C01828=1107.279,258.473,-73.640,-178.368,10.038,149.556
C01829=1107.283,258.225,-73.611,-178.370,10.036,149.556
C01830=1107.288,257.977,-73.582,-178.373,10.033,149.556
C01831=1107.291,257.728,-73.553,-178.376,10.030,149.556
C01832=1107.296,257.480,-73.524,-178.379,10.027,149.556
C01833=1107.300,257.233,-73.495,-178.381,10.025,149.556
C01834=1107.305,256.984,-73.466,-178.384,10.022,149.557
C01835=1107.308,256.736,-73.437,-178.387,10.019,149.556
C01836=1107.313,256.487,-73.409,-178.390,10.016,149.557
C01837=1107.318,256.239,-73.379,-178.393,10.014,149.557
C01838=1107.322,255.991,-73.350,-178.395,10.011,149.557
C01839=1107.325,255.742,-73.322,-178.397,10.009,149.557
C01840=1107.331,255.398,-73.282,-178.401,10.005,149.557
C01841=1107.338,255.055,-73.242,-178.405,10.001,149.557
C01842=1107.343,254.711,-73.202,-178.409,9.998,149.557
C01843=1107.349,254.367,-73.162,-178.413,9.994,149.557
C01844=1107.353,254.119,-73.133,-178.415,9.992,149.557
C01845=1107.358,253.871,-73.105,-178.418,9.989,149.557
C01846=1107.362,253.623,-73.075,-178.421,9.987,149.558
C01847=1107.366,253.374,-73.047,-178.423,9.985,149.558
C01848=1107.371,253.127,-73.018,-178.427,9.982,149.558
C01849=1107.375,252.878,-72.989,-178.429,9.979,149.558
C01850=1107.379,252.629,-72.961,-178.432,9.977,149.558
C01851=1107.383,252.381,-72.932,-178.435,9.975,149.558
C01852=1107.387,252.133,-72.904,-178.438,9.972,149.558
C01853=1107.392,251.885,-72.875,-178.440,9.970,149.559
C01854=1107.396,251.636,-72.846,-178.443,9.968,149.559
C01855=1107.400,251.388,-72.818,-178.446,9.965,149.559
C01856=1107.405,251.140,-72.789,-178.449,9.963,149.559
C01857=1107.408,250.891,-72.760,-178.452,9.960,149.559
C01858=1107.413,250.643,-72.732,-178.455,9.958,149.560
C01859=1107.417,250.394,-72.704,-178.458,9.955,149.560
C01860=1107.421,250.146,-72.675,-178.460,9.953,149.560
C01861=1107.426,249.898,-72.647,-178.463,9.950,149.560
C01862=1107.430,249.649,-72.618,-178.466,9.947,149.560
C01863=1107.435,249.401,-72.590,-178.469,9.945,149.560
C01864=1107.439,249.153,-72.561,-178.472,9.942,149.560
C01865=1107.443,248.905,-72.533,-178.474,9.940,149.560
C01866=1107.448,248.656,-72.504,-178.477,9.937,149.560
C01867=1107.451,248.408,-72.476,-178.480,9.934,149.560
C01868=1107.456,248.159,-72.447,-178.483,9.931,149.561
C01869=1107.460,247.911,-72.420,-178.485,9.928,149.560
C01870=1107.464,247.663,-72.390,-178.488,9.925,149.561
C01871=1107.469,247.415,-72.362,-178.491,9.922,149.560
C01872=1107.473,247.166,-72.334,-178.493,9.919,149.560
C01873=1107.477,246.917,-72.306,-178.496,9.916,149.560
C01874=1107.481,246.670,-72.278,-178.499,9.913,149.560
C01875=1107.486,246.421,-72.249,-178.501,9.910,149.560
C01876=1107.490,246.173,-72.221,-178.503,9.908,149.560
C01877=1107.494,245.924,-72.193,-178.506,9.905,149.560
C01878=1107.499,245.676,-72.165,-178.509,9.902,149.560
C01879=1107.503,245.428,-72.137,-178.511,9.899,149.560
C01880=1107.508,245.179,-72.108,-178.513,9.897,149.560
C01881=1107.512,244.931,-72.080,-178.516,9.894,149.560
C01882=1107.516,244.683,-72.052,-178.519,9.891,149.560
C01883=1107.520,244.434,-72.024,-178.521,9.888,149.560
C01884=1107.524,244.185,-71.995,-178.524,9.886,149.560
C01885=1107.529,243.938,-71.968,-178.527,9.883,149.561
C01886=1107.533,243.689,-71.939,-178.529,9.880,149.560
C01887=1107.537,243.441,-71.911,-178.532,9.877,149.561
C01888=1107.541,243.192,-71.883,-178.534,9.875,149.561
C01889=1107.545,242.944,-71.855,-178.537,9.872,149.561
C01890=1107.550,242.695,-71.827,-178.540,9.870,149.561
C01891=1107.555,242.447,-71.799,-178.542,9.867,149.561
C01892=1107.558,242.235,-71.775,-178.545,9.864,149.561
C01893=1107.562,242.022,-71.752,-178.547,9.862,149.561
C01894=1107.565,241.809,-71.727,-178.549,9.860,149.561
C01895=1107.569,241.597,-71.703,-178.551,9.858,149.561
C01896=1107.572,241.384,-71.680,-178.553,9.856,149.561
C01897=1107.577,241.171,-71.655,-178.555,9.854,149.561
C01898=1107.581,240.959,-71.632,-178.558,9.851,149.561
C01899=1107.584,240.746,-71.608,-178.560,9.849,149.561
C01900=1107.588,240.498,-71.579,-178.563,9.847,149.561
C01901=1107.593,240.249,-71.552,-178.565,9.844,149.561
C01902=1107.596,240.001,-71.524,-178.568,9.841,149.561
C01903=1107.602,239.752,-71.496,-178.570,9.839,149.562
C01904=1107.606,239.503,-71.468,-178.573,9.836,149.562
C01905=1107.610,239.255,-71.441,-178.576,9.833,149.562
C01906=1107.614,239.008,-71.413,-178.579,9.830,149.562
C01907=1107.618,238.759,-71.385,-178.581,9.828,149.562
C01908=1107.623,238.510,-71.358,-178.584,9.826,149.562
C01909=1107.626,238.262,-71.329,-178.587,9.823,149.562
C01910=1107.632,238.013,-71.302,-178.589,9.821,149.562
C01911=1107.636,237.765,-71.274,-178.592,9.818,149.562
C01912=1107.640,237.517,-71.246,-178.595,9.815,149.562
C01913=1107.645,237.268,-71.219,-178.597,9.813,149.562
C01914=1107.648,237.020,-71.191,-178.600,9.810,149.562
C01915=1107.653,236.771,-71.164,-178.603,9.807,149.562
C01916=1107.657,236.523,-71.136,-178.605,9.805,149.563
C01917=1107.661,236.275,-71.108,-178.608,9.802,149.563
C01918=1107.666,236.026,-71.081,-178.611,9.800,149.563
C01919=1107.670,235.778,-71.053,-178.613,9.797,149.563
C01920=1107.674,235.529,-71.025,-178.616,9.795,149.563
C01921=1107.679,235.281,-70.998,-178.619,9.792,149.563
C01922=1107.683,235.033,-70.971,-178.621,9.789,149.563
C01923=1107.687,234.784,-70.942,-178.623,9.787,149.563
C01924=1107.692,234.536,-70.915,-178.626,9.784,149.563
C01925=1107.696,234.287,-70.888,-178.629,9.781,149.563
C01926=1107.700,234.039,-70.860,-178.631,9.779,149.563
C01927=1107.705,233.790,-70.833,-178.634,9.776,149.563
C01928=1107.709,233.542,-70.805,-178.637,9.773,149.563
C01929=1107.713,233.293,-70.778,-178.640,9.771,149.564
C01930=1107.717,233.045,-70.750,-178.642,9.768,149.564
C01931=1107.722,232.797,-70.723,-178.645,9.766,149.564
C01932=1107.726,232.547,-70.696,-178.647,9.763,149.564
C01933=1107.730,232.300,-70.668,-178.650,9.760,149.564
C01934=1107.735,232.051,-70.641,-178.653,9.758,149.564
C01935=1107.740,231.803,-70.614,-178.655,9.755,149.564
C01936=1107.744,231.554,-70.586,-178.658,9.752,149.564
C01937=1107.748,231.305,-70.559,-178.661,9.749,149.564
C01938=1107.753,231.057,-70.532,-178.663,9.747,149.564
C01939=1107.758,230.808,-70.504,-178.665,9.744,149.564
C01940=1107.761,230.560,-70.477,-178.668,9.741,149.564
C01941=1107.765,230.312,-70.450,-178.671,9.738,149.564
C01942=1107.770,230.063,-70.423,-178.674,9.735,149.564
C01943=1107.774,229.815,-70.396,-178.676,9.733,149.564
C01944=1107.778,229.566,-70.368,-178.679,9.730,149.564
C01945=1107.783,229.318,-70.341,-178.681,9.727,149.564
C01946=1107.788,229.069,-70.313,-178.684,9.724,149.564
C01947=1107.791,228.821,-70.287,-178.687,9.721,149.564
C01948=1107.795,228.608,-70.263,-178.689,9.719,149.564
C01949=1107.799,228.395,-70.240,-178.690,9.716,149.564
C01950=1107.803,228.183,-70.217,-178.693,9.714,149.564
C01951=1107.806,227.970,-70.194,-178.695,9.711,149.564
C01952=1107.810,227.757,-70.170,-178.697,9.709,149.564
C01953=1107.814,227.545,-70.147,-178.700,9.706,149.564
C01954=1107.817,227.332,-70.124,-178.702,9.704,149.564
C01955=1107.821,227.119,-70.101,-178.704,9.702,149.564
C01956=1107.826,226.870,-70.074,-178.706,9.699,149.564
C01957=1107.830,226.622,-70.047,-178.709,9.695,149.564
C01958=1107.834,226.374,-70.020,-178.712,9.692,149.564
C01959=1107.838,226.124,-69.993,-178.714,9.689,149.564
C01960=1107.843,225.876,-69.966,-178.716,9.687,149.564
C01961=1107.848,225.627,-69.939,-178.718,9.684,149.564
C01962=1107.852,225.379,-69.912,-178.721,9.681,149.564
C01963=1107.856,225.131,-69.885,-178.723,9.678,149.564
C01964=1107.861,224.882,-69.858,-178.726,9.674,149.563
C01965=1107.865,224.634,-69.832,-178.729,9.671,149.563
C01966=1107.869,224.386,-69.805,-178.731,9.668,149.563
C01967=1107.874,224.136,-69.778,-178.733,9.666,149.563
C01968=1107.878,223.888,-69.751,-178.735,9.663,149.563
C01969=1107.882,223.639,-69.724,-178.738,9.660,149.563
C01970=1107.887,223.391,-69.697,-178.741,9.657,149.563
C01971=1107.891,223.142,-69.671,-178.743,9.653,149.563
C01972=1107.896,222.894,-69.644,-178.746,9.650,149.563
C01973=1107.900,222.646,-69.617,-178.748,9.647,149.563
C01974=1107.904,222.397,-69.590,-178.750,9.645,149.563
C01975=1107.909,222.148,-69.564,-178.753,9.642,149.563
C01976=1107.913,221.900,-69.537,-178.755,9.639,149.563
C01977=1107.918,221.651,-69.510,-178.757,9.635,149.562
C01978=1107.922,221.403,-69.484,-178.760,9.632,149.562
C01979=1107.926,221.155,-69.457,-178.762,9.629,149.562
C01980=1107.931,220.905,-69.430,-178.765,9.626,149.562
C01981=1107.935,220.657,-69.404,-178.767,9.623,149.562
C01982=1107.939,220.408,-69.377,-178.769,9.620,149.562
C01983=1107.943,220.160,-69.350,-178.771,9.617,149.562
C01984=1107.948,219.911,-69.324,-178.774,9.614,149.562
C01985=1107.952,219.663,-69.297,-178.776,9.611,149.562
C01986=1107.957,219.414,-69.270,-178.779,9.608,149.562
C01987=1107.961,219.166,-69.245,-178.781,9.605,149.562
C01988=1107.966,218.917,-69.217,-178.783,9.602,149.561
C01989=1107.970,218.669,-69.191,-178.785,9.599,149.561
C01990=1107.974,218.420,-69.165,-178.788,9.596,149.561
C01991=1107.978,218.172,-69.138,-178.790,9.592,149.561
C01992=1107.982,217.923,-69.112,-178.793,9.589,149.561
C01993=1107.987,217.674,-69.085,-178.794,9.587,149.561
C01994=1107.991,217.426,-69.059,-178.797,9.583,149.561
C01995=1107.996,217.177,-69.033,-178.799,9.580,149.561
C01996=1108.000,216.929,-69.006,-178.802,9.577,149.561
C01997=1108.005,216.680,-68.980,-178.803,9.575,149.560
C01998=1108.009,216.431,-68.953,-178.806,9.571,149.560
C01999=1108.013,216.183,-68.928,-178.808,9.568,149.560
C02000=1108.018,215.935,-68.901,-178.811,9.565,149.560
C02001=1108.023,215.686,-68.875,-178.814,9.562,149.560
C02002=1108.027,215.438,-68.848,-178.815,9.559,149.560
C02003=1108.032,215.189,-68.822,-178.818,9.556,149.560
C02004=1108.035,214.976,-68.799,-178.819,9.554,149.560
C02005=1108.039,214.763,-68.777,-178.821,9.552,149.560
C02006=1108.042,214.550,-68.755,-178.824,9.549,149.560
C02007=1108.046,214.338,-68.732,-178.826,9.546,149.560
C02008=1108.050,214.124,-68.709,-178.827,9.544,149.559
C02009=1108.054,213.912,-68.688,-178.829,9.541,149.559
C02010=1108.057,213.699,-68.665,-178.831,9.539,149.559
C02011=1108.062,213.486,-68.642,-178.834,9.536,149.559
C02012=1108.066,213.237,-68.617,-178.836,9.533,149.559
C02013=1108.070,212.989,-68.590,-178.840,9.529,149.559
C02014=1108.075,212.740,-68.564,-178.842,9.526,149.559
C02015=1108.079,212.491,-68.538,-178.846,9.522,149.559
C02016=1108.083,212.243,-68.511,-178.849,9.520,149.559
C02017=1108.087,211.994,-68.486,-178.852,9.516,149.559
C02018=1108.093,211.746,-68.460,-178.855,9.513,149.559
C02019=1108.097,211.497,-68.433,-178.858,9.509,149.559
C02020=1108.101,211.249,-68.408,-178.861,9.506,149.559
C02021=1108.105,211.000,-68.382,-178.864,9.503,149.560
C02022=1108.110,210.751,-68.355,-178.867,9.500,149.560
C02023=1108.114,210.502,-68.329,-178.871,9.496,149.560
C02024=1108.119,210.254,-68.304,-178.873,9.494,149.560
C02025=1108.123,210.006,-68.278,-178.876,9.491,149.560
C02026=1108.127,209.757,-68.252,-178.880,9.487,149.560
C02027=1108.131,209.508,-68.226,-178.883,9.484,149.560
C02028=1108.136,209.259,-68.200,-178.885,9.481,149.560
C02029=1108.141,209.011,-68.174,-178.889,9.478,149.560
C02030=1108.145,208.763,-68.148,-178.892,9.475,149.560
C02031=1108.149,208.514,-68.122,-178.895,9.472,149.560
C02032=1108.154,208.265,-68.097,-178.897,9.469,149.561
C02033=1108.158,208.017,-68.071,-178.901,9.466,149.561
C02034=1108.163,207.768,-68.045,-178.904,9.463,149.561
C02035=1108.167,207.519,-68.020,-178.907,9.460,149.561
C02036=1108.172,207.270,-67.993,-178.909,9.457,149.561
C02037=1108.177,207.022,-67.968,-178.912,9.454,149.561
C02038=1108.181,206.773,-67.942,-178.915,9.451,149.561
C02039=1108.185,206.524,-67.917,-178.919,9.448,149.561
C02040=1108.189,206.276,-67.891,-178.921,9.445,149.561
C02041=1108.194,206.027,-67.865,-178.924,9.442,149.561
C02042=1108.198,205.779,-67.840,-178.927,9.439,149.561
C02043=1108.203,205.530,-67.814,-178.930,9.436,149.561
C02044=1108.207,205.282,-67.788,-178.933,9.434,149.562
C02045=1108.212,205.033,-67.763,-178.936,9.431,149.562
C02046=1108.216,204.784,-67.738,-178.938,9.428,149.562
C02047=1108.221,204.535,-67.712,-178.941,9.425,149.562
C02048=1108.225,204.287,-67.687,-178.944,9.422,149.562
C02049=1108.229,204.038,-67.661,-178.947,9.420,149.562
C02050=1108.234,203.790,-67.635,-178.950,9.417,149.562
C02051=1108.239,203.541,-67.610,-178.953,9.414,149.562
C02052=1108.243,203.291,-67.585,-178.956,9.411,149.562
C02053=1108.248,203.043,-67.559,-178.958,9.408,149.562
C02054=1108.252,202.795,-67.534,-178.961,9.405,149.562
C02055=1108.256,202.546,-67.508,-178.964,9.402,149.563
C02056=1108.260,202.298,-67.483,-178.967,9.399,149.562
C02057=1108.265,202.049,-67.458,-178.970,9.397,149.563
C02058=1108.269,201.800,-67.432,-178.972,9.393,149.563
C02059=1108.274,201.552,-67.407,-178.975,9.391,149.563
C02060=1108.278,201.338,-67.386,-178.977,9.388,149.563
C02061=1108.281,201.125,-67.363,-178.979,9.386,149.563
C02062=1108.285,200.912,-67.342,-178.982,9.383,149.563
C02063=1108.290,200.699,-67.321,-178.984,9.381,149.563
C02064=1108.293,200.486,-67.298,-178.986,9.379,149.563
C02065=1108.297,200.273,-67.277,-178.988,9.376,149.563
C02066=1108.301,200.060,-67.255,-178.990,9.374,149.563
C02067=1108.304,199.848,-67.234,-178.993,9.372,149.563
C02068=1108.308,199.599,-67.208,-178.995,9.368,149.563
C02069=1108.314,199.350,-67.184,-178.998,9.365,149.563
C02070=1108.318,199.101,-67.158,-179.001,9.363,149.563
C02071=1108.322,198.852,-67.133,-179.003,9.360,149.563
C02072=1108.326,198.604,-67.108,-179.006,9.356,149.563
C02073=1108.331,198.355,-67.083,-179.008,9.353,149.563
C02074=1108.336,198.107,-67.058,-179.010,9.351,149.563
C02075=1108.340,197.857,-67.033,-179.013,9.348,149.563
C02076=1108.344,197.609,-67.008,-179.016,9.345,149.563
C02077=1108.349,197.360,-66.983,-179.018,9.342,149.563
C02078=1108.354,197.112,-66.958,-179.021,9.339,149.563
C02079=1108.358,196.862,-66.932,-179.023,9.336,149.563
C02080=1108.362,196.615,-66.908,-179.025,9.333,149.563
C02081=1108.367,196.365,-66.883,-179.027,9.330,149.562
C02082=1108.372,196.117,-66.857,-179.030,9.327,149.562
C02083=1108.375,195.868,-66.833,-179.032,9.325,149.562
C02084=1108.380,195.620,-66.807,-179.034,9.321,149.562
C02085=1108.385,195.370,-66.782,-179.036,9.318,149.562
C02086=1108.389,195.122,-66.758,-179.038,9.316,149.562
C02087=1108.393,194.873,-66.733,-179.041,9.313,149.562
C02088=1108.399,194.625,-66.708,-179.043,9.310,149.562
C02089=1108.402,194.375,-66.683,-179.045,9.307,149.562
C02090=1108.407,194.127,-66.658,-179.047,9.304,149.562
C02091=1108.411,193.878,-66.634,-179.049,9.301,149.562
C02092=1108.416,193.629,-66.609,-179.052,9.298,149.561
C02093=1108.420,193.381,-66.583,-179.053,9.296,149.561
C02094=1108.425,193.132,-66.559,-179.056,9.293,149.561
C02095=1108.430,192.884,-66.534,-179.058,9.290,149.561
C02096=1108.433,192.635,-66.509,-179.060,9.287,149.561
C02097=1108.438,192.386,-66.485,-179.063,9.284,149.561
C02098=1108.443,192.137,-66.460,-179.065,9.282,149.561
C02099=1108.447,191.888,-66.436,-179.067,9.279,149.561
C02100=1108.452,191.639,-66.411,-179.069,9.276,149.561
C02101=1108.456,191.391,-66.386,-179.071,9.273,149.561
C02102=1108.461,191.143,-66.361,-179.074,9.270,149.561
C02103=1108.465,190.893,-66.337,-179.076,9.267,149.561
C02104=1108.470,190.645,-66.312,-179.078,9.264,149.561
C02105=1108.474,190.396,-66.288,-179.080,9.262,149.561
C02106=1108.479,190.148,-66.262,-179.083,9.259,149.561
C02107=1108.483,189.899,-66.238,-179.085,9.256,149.561
C02108=1108.488,189.650,-66.213,-179.087,9.253,149.561
C02109=1108.492,189.401,-66.189,-179.090,9.250,149.561
C02110=1108.497,189.153,-66.164,-179.092,9.247,149.560
C02111=1108.501,188.903,-66.140,-179.094,9.245,149.560
C02112=1108.506,188.655,-66.115,-179.097,9.242,149.560
C02113=1108.510,188.406,-66.091,-179.098,9.239,149.560
C02114=1108.515,188.157,-66.066,-179.101,9.236,149.560
C02115=1108.519,187.908,-66.042,-179.104,9.234,149.560
C02116=1108.524,187.695,-66.021,-179.106,9.231,149.560
C02117=1108.527,187.483,-66.000,-179.108,9.229,149.560
C02118=1108.531,187.270,-65.979,-179.110,9.227,149.560
C02119=1108.535,187.056,-65.957,-179.111,9.224,149.560
C02120=1108.539,186.843,-65.937,-179.113,9.222,149.560
C02121=1108.543,186.630,-65.916,-179.115,9.220,149.560
C02122=1108.546,186.417,-65.895,-179.117,9.217,149.560
C02123=1108.551,186.204,-65.874,-179.120,9.214,149.560
C02124=1108.554,185.955,-65.850,-179.122,9.212,149.560
C02125=1108.559,185.706,-65.825,-179.124,9.209,149.560
C02126=1108.564,185.458,-65.801,-179.126,9.206,149.560
C02127=1108.568,185.209,-65.777,-179.128,9.203,149.560
C02128=1108.573,184.959,-65.753,-179.131,9.200,149.560
C02129=1108.577,184.711,-65.728,-179.134,9.197,149.560
C02130=1108.582,184.462,-65.704,-179.135,9.195,149.560
C02131=1108.586,184.213,-65.679,-179.138,9.192,149.560
C02132=1108.591,183.965,-65.655,-179.140,9.189,149.560
C02133=1108.595,183.716,-65.631,-179.142,9.186,149.560
C02134=1108.600,183.468,-65.607,-179.145,9.183,149.560
C02135=1108.604,183.218,-65.583,-179.147,9.180,149.560
C02136=1108.609,182.969,-65.559,-179.149,9.178,149.560
C02137=1108.614,182.721,-65.534,-179.151,9.174,149.559
C02138=1108.618,182.472,-65.510,-179.154,9.171,149.559
C02139=1108.622,182.223,-65.486,-179.156,9.168,149.559
C02140=1108.627,181.974,-65.462,-179.158,9.166,149.559
C02141=1108.632,181.725,-65.438,-179.161,9.162,149.559
C02142=1108.636,181.477,-65.413,-179.163,9.159,149.559
C02143=1108.641,181.229,-65.389,-179.166,9.156,149.559
C02144=1108.645,180.979,-65.366,-179.168,9.154,149.559
C02145=1108.649,180.730,-65.342,-179.170,9.151,149.559
C02146=1108.654,180.482,-65.317,-179.173,9.148,149.559
C02147=1108.659,180.233,-65.294,-179.175,9.144,149.559
C02148=1108.663,179.984,-65.269,-179.177,9.142,149.559
C02149=1108.667,179.735,-65.245,-179.179,9.139,149.559
C02150=1108.672,179.486,-65.222,-179.182,9.136,149.559
C02151=1108.676,179.238,-65.198,-179.184,9.132,149.558
C02152=1108.681,178.989,-65.173,-179.186,9.130,149.558
C02153=1108.686,178.740,-65.150,-179.188,9.127,149.558
C02154=1108.691,178.492,-65.126,-179.191,9.124,149.558
C02155=1108.695,178.242,-65.102,-179.192,9.121,149.558
C02156=1108.699,177.993,-65.078,-179.195,9.118,149.558
C02157=1108.703,177.745,-65.054,-179.197,9.115,149.558
C02158=1108.708,177.496,-65.030,-179.199,9.112,149.558
C02159=1108.713,177.248,-65.006,-179.201,9.109,149.558
C02160=1108.717,176.998,-64.983,-179.204,9.106,149.558
C02161=1108.722,176.750,-64.959,-179.205,9.103,149.557
C02162=1108.727,176.500,-64.934,-179.208,9.100,149.557
C02163=1108.731,176.252,-64.910,-179.210,9.097,149.557
C02164=1108.736,176.003,-64.887,-179.212,9.094,149.557
C02165=1108.740,175.754,-64.863,-179.214,9.091,149.557
C02166=1108.745,175.505,-64.840,-179.217,9.088,149.557
C02167=1108.749,175.256,-64.816,-179.218,9.085,149.557
C02168=1108.754,175.008,-64.792,-179.221,9.082,149.557
C02169=1108.758,174.759,-64.769,-179.223,9.079,149.557
C02170=1108.763,174.510,-64.745,-179.225,9.076,149.556
C02171=1108.768,174.261,-64.721,-179.227,9.073,149.556
C02172=1108.771,174.048,-64.701,-179.229,9.071,149.556
C02173=1108.775,173.835,-64.681,-179.231,9.068,149.556
C02174=1108.779,173.621,-64.660,-179.233,9.066,149.556
C02175=1108.783,173.408,-64.640,-179.235,9.064,149.556
C02176=1108.786,173.195,-64.620,-179.237,9.060,149.556
C02177=1108.791,172.982,-64.600,-179.239,9.058,149.556
C02178=1108.795,172.768,-64.580,-179.240,9.055,149.556
C02179=1108.799,172.555,-64.559,-179.242,9.053,149.556
C02180=1108.803,172.306,-64.536,-179.244,9.050,149.555
C02181=1108.808,172.058,-64.512,-179.246,9.047,149.555
C02182=1108.812,171.809,-64.488,-179.249,9.044,149.555
C02183=1108.816,171.560,-64.466,-179.251,9.041,149.555
C02184=1108.821,171.311,-64.442,-179.253,9.038,149.555
C02185=1108.825,171.063,-64.418,-179.255,9.035,149.555
C02186=1108.830,170.814,-64.395,-179.257,9.032,149.555
C02187=1108.835,170.565,-64.372,-179.259,9.029,149.555
C02188=1108.840,170.316,-64.348,-179.262,9.026,149.555
C02189=1108.844,170.067,-64.325,-179.264,9.023,149.554
C02190=1108.849,169.818,-64.301,-179.266,9.020,149.554
C02191=1108.853,169.569,-64.277,-179.268,9.017,149.554
C02192=1108.857,169.320,-64.255,-179.270,9.014,149.554
C02193=1108.862,169.071,-64.231,-179.272,9.012,149.554
C02194=1108.867,168.822,-64.208,-179.275,9.008,149.554
C02195=1108.871,168.573,-64.185,-179.277,9.005,149.554
C02196=1108.876,168.324,-64.161,-179.279,9.003,149.554
C02197=1108.881,168.076,-64.137,-179.281,8.999,149.554
C02198=1108.884,167.827,-64.114,-179.283,8.996,149.553
C02199=1108.889,167.578,-64.091,-179.285,8.994,149.553
C02200=1108.894,167.329,-64.068,-179.287,8.990,149.553
C02201=1108.899,167.081,-64.045,-179.290,8.987,149.553
C02202=1108.904,166.832,-64.021,-179.291,8.984,149.553
C02203=1108.908,166.583,-63.999,-179.294,8.981,149.553
C02204=1108.913,166.334,-63.975,-179.296,8.978,149.553
C02205=1108.917,166.085,-63.952,-179.298,8.975,149.553
C02206=1108.922,165.836,-63.928,-179.300,8.972,149.553
C02207=1108.926,165.587,-63.906,-179.302,8.969,149.552
C02208=1108.931,165.338,-63.882,-179.305,8.966,149.552
C02209=1108.935,165.089,-63.859,-179.306,8.963,149.552
C02210=1108.941,164.841,-63.836,-179.309,8.960,149.552
C02211=1108.945,164.592,-63.813,-179.311,8.956,149.552
C02212=1108.949,164.343,-63.790,-179.314,8.953,149.552
C02213=1108.954,164.094,-63.767,-179.315,8.951,149.552
C02214=1108.958,163.845,-63.744,-179.318,8.947,149.551
C02215=1108.963,163.596,-63.721,-179.320,8.944,149.551
C02216=1108.968,163.347,-63.698,-179.321,8.942,149.551
C02217=1108.972,163.098,-63.675,-179.324,8.939,149.551
C02218=1108.977,162.850,-63.652,-179.326,8.935,149.551
C02219=1108.982,162.600,-63.629,-179.329,8.932,149.551
C02220=1108.986,162.352,-63.606,-179.330,8.929,149.551
C02221=1108.991,162.102,-63.583,-179.333,8.926,149.551
C02222=1108.995,161.853,-63.560,-179.335,8.923,149.550
C02223=1108.999,161.604,-63.537,-179.337,8.920,149.550
C02224=1109.005,161.356,-63.514,-179.339,8.917,149.550
C02225=1109.009,161.107,-63.491,-179.341,8.913,149.550
C02226=1109.014,160.858,-63.469,-179.343,8.910,149.550
C02227=1109.017,160.609,-63.446,-179.345,8.907,149.550
C02228=1109.022,160.396,-63.426,-179.347,8.904,149.550
C02229=1109.026,160.183,-63.407,-179.349,8.902,149.549
C02230=1109.029,159.969,-63.387,-179.351,8.899,149.549
C02231=1109.034,159.756,-63.367,-179.352,8.897,149.549
C02232=1109.038,159.543,-63.348,-179.355,8.894,149.549
C02233=1109.041,159.329,-63.328,-179.356,8.891,149.549
C02234=1109.045,159.116,-63.309,-179.358,8.889,149.549
C02235=1109.049,158.902,-63.290,-179.359,8.886,149.549
C02236=1109.054,158.653,-63.267,-179.362,8.883,149.549
C02237=1109.058,158.405,-63.244,-179.364,8.879,149.548
C02238=1109.063,158.156,-63.222,-179.366,8.876,149.548
C02239=1109.067,157.907,-63.199,-179.369,8.873,149.548
C02240=1109.072,157.658,-63.175,-179.370,8.870,149.548
C02241=1109.077,157.409,-63.154,-179.372,8.866,149.548
C02242=1109.082,157.160,-63.130,-179.375,8.863,149.547
C02243=1109.086,156.911,-63.108,-179.377,8.860,149.547
C02244=1109.091,156.662,-63.085,-179.379,8.856,149.547
C02245=1109.095,156.413,-63.063,-179.380,8.854,149.547
C02246=1109.100,156.164,-63.040,-179.383,8.851,149.547
C02247=1109.104,155.915,-63.017,-179.385,8.847,149.547
C02248=1109.109,155.667,-62.995,-179.387,8.844,149.546
C02249=1109.114,155.418,-62.972,-179.389,8.840,149.546
C02250=1109.118,155.168,-62.950,-179.391,8.838,149.546
C02251=1109.123,154.920,-62.927,-179.393,8.834,149.546
C02252=1109.127,154.671,-62.905,-179.395,8.831,149.546
C02253=1109.132,154.421,-62.883,-179.397,8.827,149.545
C02254=1109.137,154.173,-62.860,-179.399,8.824,149.545
C02255=1109.141,153.924,-62.838,-179.402,8.821,149.545
C02256=1109.146,153.675,-62.815,-179.403,8.818,149.545
C02257=1109.151,153.426,-62.793,-179.405,8.814,149.545
C02258=1109.155,153.177,-62.770,-179.407,8.811,149.544
C02259=1109.160,152.928,-62.747,-179.409,8.807,149.544
C02260=1109.165,152.679,-62.726,-179.412,8.804,149.544
C02261=1109.169,152.430,-62.703,-179.414,8.801,149.544
C02262=1109.174,152.181,-62.681,-179.416,8.797,149.544
C02263=1109.179,151.932,-62.659,-179.418,8.794,149.543
C02264=1109.182,151.683,-62.636,-179.420,8.791,149.543
C02265=1109.187,151.435,-62.614,-179.422,8.788,149.543
C02266=1109.192,151.185,-62.592,-179.424,8.784,149.543
C02267=1109.196,150.936,-62.569,-179.426,8.781,149.542
C02268=1109.201,150.688,-62.547,-179.428,8.777,149.542
C02269=1109.206,150.438,-62.525,-179.430,8.774,149.542
C02270=1109.211,150.189,-62.503,-179.432,8.770,149.542
C02271=1109.215,149.941,-62.480,-179.434,8.767,149.541
C02272=1109.220,149.692,-62.458,-179.436,8.763,149.541
C02273=1109.225,149.442,-62.436,-179.438,8.760,149.541
C02274=1109.230,149.194,-62.414,-179.440,8.756,149.541
C02275=1109.234,148.944,-62.392,-179.442,8.752,149.540
C02276=1109.238,148.696,-62.369,-179.444,8.750,149.540
C02277=1109.243,148.447,-62.348,-179.446,8.746,149.540
C02278=1109.248,148.197,-62.325,-179.448,8.743,149.540
C02279=1109.253,147.949,-62.303,-179.450,8.739,149.539
C02280=1109.257,147.699,-62.281,-179.452,8.736,149.539
C02281=1109.262,147.451,-62.260,-179.454,8.732,149.539
C02282=1109.266,147.201,-62.237,-179.456,8.729,149.539
C02283=1109.271,146.953,-62.215,-179.458,8.725,149.538
C02284=1109.275,146.739,-62.196,-179.460,8.721,149.538
C02285=1109.279,146.526,-62.178,-179.461,8.719,149.538
C02286=1109.283,146.312,-62.158,-179.463,8.716,149.537
C02287=1109.287,146.099,-62.139,-179.465,8.713,149.537
C02288=1109.291,145.886,-62.121,-179.466,8.710,149.537
C02289=1109.295,145.672,-62.102,-179.468,8.706,149.537
C02290=1109.299,145.459,-62.083,-179.470,8.704,149.537
C02291=1109.303,145.245,-62.064,-179.472,8.700,149.536
C02292=1109.308,144.996,-62.043,-179.473,8.697,149.536
C02293=1109.312,144.747,-62.020,-179.475,8.694,149.536
C02294=1109.317,144.498,-61.999,-179.476,8.690,149.535
C02295=1109.321,144.249,-61.977,-179.479,8.686,149.535
C02296=1109.326,144.000,-61.955,-179.480,8.683,149.535
C02297=1109.330,143.751,-61.933,-179.482,8.680,149.534
C02298=1109.335,143.502,-61.911,-179.483,8.676,149.534
C02299=1109.340,143.254,-61.890,-179.485,8.673,149.534
C02300=1109.344,143.004,-61.868,-179.486,8.669,149.533
C02301=1109.349,142.756,-61.846,-179.488,8.666,149.533
C02302=1109.354,142.506,-61.825,-179.491,8.662,149.533
C02303=1109.359,142.257,-61.803,-179.492,8.659,149.532
C02304=1109.363,142.008,-61.781,-179.494,8.656,149.532
C02305=1109.368,141.759,-61.759,-179.495,8.652,149.532
C02306=1109.373,141.510,-61.737,-179.497,8.649,149.531
C02307=1109.377,141.261,-61.715,-179.499,8.646,149.531
C02308=1109.382,141.012,-61.694,-179.500,8.642,149.531
C02309=1109.386,140.762,-61.672,-179.502,8.638,149.530
C02310=1109.391,140.514,-61.651,-179.504,8.635,149.530
C02311=1109.396,140.265,-61.629,-179.506,8.632,149.530
C02312=1109.400,140.016,-61.607,-179.508,8.628,149.530
C02313=1109.405,139.768,-61.586,-179.509,8.625,149.529
C02314=1109.409,139.518,-61.565,-179.511,8.622,149.529
C02315=1109.414,139.269,-61.543,-179.512,8.618,149.528
C02316=1109.419,139.020,-61.521,-179.514,8.614,149.528
C02317=1109.423,138.771,-61.499,-179.516,8.611,149.528
C02318=1109.428,138.522,-61.478,-179.518,8.608,149.528
C02319=1109.433,138.273,-61.457,-179.520,8.604,149.527
C02320=1109.437,138.024,-61.434,-179.521,8.601,149.527
C02321=1109.443,137.774,-61.414,-179.523,8.598,149.527
C02322=1109.447,137.526,-61.392,-179.525,8.594,149.526
C02323=1109.451,137.277,-61.370,-179.526,8.591,149.526
C02324=1109.456,137.028,-61.349,-179.528,8.587,149.526
C02325=1109.461,136.779,-61.328,-179.530,8.584,149.525
C02326=1109.465,136.530,-61.306,-179.531,8.581,149.525
C02327=1109.470,136.280,-61.285,-179.533,8.577,149.525
C02328=1109.475,136.032,-61.264,-179.535,8.574,149.525
C02329=1109.479,135.782,-61.242,-179.537,8.570,149.524
C02330=1109.484,135.533,-61.221,-179.538,8.567,149.524
C02331=1109.489,135.285,-61.199,-179.540,8.564,149.524
C02332=1109.494,135.035,-61.178,-179.542,8.560,149.523
C02333=1109.498,134.786,-61.157,-179.544,8.558,149.523
C02334=1109.503,134.537,-61.136,-179.545,8.554,149.523
C02335=1109.508,134.289,-61.114,-179.547,8.550,149.523
C02336=1109.512,134.039,-61.093,-179.549,8.548,149.522
C02337=1109.516,133.790,-61.071,-179.550,8.544,149.522
C02338=1109.522,133.541,-61.050,-179.553,8.540,149.522
C02339=1109.526,133.292,-61.029,-179.554,8.537,149.521
C02340=1109.530,133.078,-61.010,-179.556,8.534,149.521
C02341=1109.534,132.865,-60.993,-179.558,8.531,149.521
C02342=1109.538,132.652,-60.975,-179.559,8.529,149.521
C02343=1109.543,132.438,-60.956,-179.560,8.525,149.520
C02344=1109.546,132.224,-60.938,-179.561,8.523,149.520
C02345=1109.550,132.010,-60.920,-179.563,8.520,149.520
C02346=1109.554,131.797,-60.902,-179.564,8.517,149.520
C02347=1109.558,131.584,-60.884,-179.566,8.514,149.519
C02348=1109.563,131.335,-60.863,-179.568,8.511,149.519
C02349=1109.568,131.085,-60.841,-179.570,8.508,149.519
C02350=1109.572,130.837,-60.820,-179.572,8.504,149.518
C02351=1109.577,130.587,-60.800,-179.573,8.501,149.518
C02352=1109.582,130.339,-60.778,-179.575,8.498,149.518
C02353=1109.586,130.090,-60.757,-179.577,8.494,149.518
C02354=1109.591,129.840,-60.736,-179.578,8.491,149.517
C02355=1109.596,129.591,-60.714,-179.580,8.487,149.517
C02356=1109.600,129.342,-60.694,-179.582,8.484,149.517
C02357=1109.606,129.093,-60.673,-179.584,8.481,149.517
C02358=1109.610,128.845,-60.652,-179.585,8.477,149.516
C02359=1109.615,128.595,-60.631,-179.587,8.474,149.516
C02360=1109.619,128.345,-60.610,-179.589,8.471,149.516
C02361=1109.624,128.096,-60.589,-179.591,8.468,149.516
C02362=1109.629,127.848,-60.568,-179.592,8.464,149.515
C02363=1109.633,127.599,-60.547,-179.594,8.461,149.515
C02364=1109.638,127.350,-60.526,-179.596,8.458,149.515
C02365=1109.644,127.100,-60.505,-179.598,8.454,149.514
C02366=1109.648,126.852,-60.484,-179.600,8.450,149.514
C02367=1109.652,126.602,-60.463,-179.601,8.447,149.514
C02368=1109.657,126.353,-60.443,-179.603,8.444,149.514
C02369=1109.662,126.104,-60.422,-179.605,8.440,149.513
C02370=1109.666,125.855,-60.401,-179.606,8.437,149.513
C02371=1109.671,125.606,-60.380,-179.608,8.434,149.513
C02372=1109.676,125.357,-60.359,-179.610,8.430,149.512
C02373=1109.681,125.108,-60.338,-179.612,8.428,149.512
C02374=1109.685,124.859,-60.318,-179.613,8.424,149.512
C02375=1109.690,124.610,-60.297,-179.616,8.420,149.511
C02376=1109.694,124.360,-60.276,-179.617,8.418,149.511
C02377=1109.699,124.111,-60.256,-179.619,8.414,149.511
C02378=1109.704,123.862,-60.235,-179.621,8.410,149.511
C02379=1109.708,123.613,-60.214,-179.622,8.407,149.510
C02380=1109.713,123.364,-60.193,-179.624,8.404,149.510
C02381=1109.718,123.115,-60.173,-179.626,8.400,149.510
C02382=1109.723,122.865,-60.152,-179.627,8.397,149.509
C02383=1109.727,122.617,-60.132,-179.629,8.394,149.509
C02384=1109.732,122.368,-60.111,-179.631,8.390,149.509
C02385=1109.737,122.118,-60.090,-179.633,8.387,149.509
C02386=1109.742,121.869,-60.070,-179.634,8.384,149.508
C02387=1109.747,121.620,-60.049,-179.636,8.380,149.508
C02388=1109.751,121.371,-60.029,-179.639,8.377,149.508
C02389=1109.756,121.122,-60.008,-179.640,8.374,149.508
C02390=1109.761,120.873,-59.987,-179.642,8.370,149.507
C02391=1109.765,120.624,-59.967,-179.644,8.367,149.507
C02392=1109.770,120.375,-59.947,-179.645,8.364,149.507
C02393=1109.775,120.126,-59.926,-179.647,8.360,149.507
C02394=1109.779,119.877,-59.905,-179.649,8.357,149.506
C02395=1109.784,119.628,-59.885,-179.650,8.354,149.506
C02396=1109.788,119.414,-59.868,-179.652,8.350,149.506
C02397=1109.792,119.200,-59.850,-179.654,8.348,149.505
C02398=1109.796,118.987,-59.833,-179.655,8.345,149.505
C02399=1109.800,118.773,-59.815,-179.657,8.342,149.505
C02400=1109.804,118.559,-59.797,-179.658,8.340,149.505
C02401=1109.808,118.345,-59.779,-179.660,8.336,149.505
C02402=1109.812,118.132,-59.763,-179.662,8.333,149.504
C02403=1109.816,117.918,-59.745,-179.663,8.330,149.504
C02404=1109.820,117.669,-59.725,-179.665,8.327,149.504
C02405=1109.826,117.420,-59.704,-179.666,8.324,149.503
C02406=1109.831,117.171,-59.684,-179.668,8.320,149.503
C02407=1109.835,116.922,-59.663,-179.670,8.317,149.503
C02408=1109.840,116.673,-59.644,-179.671,8.314,149.503
C02409=1109.845,116.424,-59.623,-179.673,8.310,149.502
C02410=1109.849,116.175,-59.602,-179.675,8.307,149.502
C02411=1109.854,115.925,-59.583,-179.677,8.303,149.502
C02412=1109.859,115.676,-59.562,-179.678,8.300,149.501
C02413=1109.864,115.427,-59.541,-179.680,8.296,149.501
C02414=1109.868,115.178,-59.521,-179.682,8.293,149.501
C02415=1109.873,114.928,-59.501,-179.683,8.290,149.501
C02416=1109.877,114.679,-59.481,-179.685,8.287,149.500
C02417=1109.882,114.430,-59.461,-179.687,8.283,149.500
C02418=1109.887,114.182,-59.441,-179.689,8.279,149.500
C02419=1109.892,113.932,-59.420,-179.691,8.277,149.499
C02420=1109.897,113.683,-59.401,-179.692,8.273,149.499
C02421=1109.902,113.434,-59.380,-179.694,8.269,149.499
C02422=1109.906,113.185,-59.360,-179.696,8.266,149.499
C02423=1109.911,112.935,-59.340,-179.697,8.263,149.498
C02424=1109.915,112.686,-59.320,-179.699,8.259,149.498
C02425=1109.921,112.438,-59.301,-179.701,8.255,149.497
C02426=1109.926,112.188,-59.280,-179.703,8.252,149.497
C02427=1109.930,111.939,-59.260,-179.704,8.249,149.497
C02428=1109.935,111.690,-59.240,-179.706,8.245,149.497
C02429=1109.940,111.440,-59.220,-179.708,8.242,149.496
C02430=1109.944,111.191,-59.200,-179.710,8.238,149.496
C02431=1109.949,110.942,-59.180,-179.711,8.235,149.496
C02432=1109.954,110.693,-59.160,-179.713,8.232,149.495
C02433=1109.959,110.444,-59.140,-179.716,8.227,149.495
C02434=1109.963,110.195,-59.120,-179.718,8.224,149.495
C02435=1109.968,109.945,-59.100,-179.720,8.220,149.495
C02436=1109.973,109.697,-59.080,-179.722,8.216,149.494
C02437=1109.978,109.447,-59.061,-179.724,8.213,149.494
C02438=1109.982,109.199,-59.040,-179.725,8.209,149.494
C02439=1109.987,108.949,-59.021,-179.727,8.205,149.493
C02440=1109.992,108.700,-59.001,-179.729,8.202,149.493
C02441=1109.997,108.451,-58.981,-179.731,8.198,149.493
C02442=1110.001,108.202,-58.961,-179.733,8.195,149.493
C02443=1110.006,107.952,-58.942,-179.735,8.191,149.492
C02444=1110.010,107.703,-58.921,-179.737,8.187,149.492
C02445=1110.016,107.454,-58.902,-179.739,8.184,149.492
C02446=1110.021,107.205,-58.882,-179.740,8.180,149.491
C02447=1110.025,106.956,-58.862,-179.742,8.176,149.491
C02448=1110.030,106.707,-58.843,-179.744,8.172,149.491
C02449=1110.035,106.457,-58.823,-179.746,8.169,149.490
C02450=1110.039,106.208,-58.803,-179.748,8.165,149.490
C02451=1110.044,105.959,-58.783,-179.750,8.162,149.490
C02452=1110.048,105.745,-58.766,-179.751,8.159,149.489
C02453=1110.053,105.532,-58.750,-179.753,8.155,149.489
C02454=1110.056,105.318,-58.733,-179.754,8.152,149.489
C02455=1110.061,105.104,-58.716,-179.756,8.149,149.489
C02456=1110.064,104.890,-58.700,-179.757,8.146,149.488
C02457=1110.069,104.676,-58.682,-179.759,8.143,149.488
C02458=1110.073,104.462,-58.666,-179.761,8.139,149.488
C02459=1110.077,104.249,-58.649,-179.762,8.136,149.487
C02460=1110.082,104.000,-58.629,-179.764,8.133,149.487
C02461=1110.086,103.750,-58.610,-179.765,8.129,149.487
C02462=1110.091,103.501,-58.590,-179.767,8.125,149.486
C02463=1110.096,103.253,-58.571,-179.769,8.121,149.486
C02464=1110.101,103.003,-58.551,-179.771,8.118,149.485
C02465=1110.106,102.754,-58.532,-179.772,8.114,149.485
C02466=1110.110,102.505,-58.513,-179.774,8.110,149.485
C02467=1110.115,102.255,-58.493,-179.776,8.106,149.484
C02468=1110.120,102.006,-58.474,-179.778,8.102,149.484
C02469=1110.125,101.757,-58.454,-179.779,8.099,149.484
C02470=1110.130,101.507,-58.434,-179.780,8.095,149.483
C02471=1110.134,101.259,-58.416,-179.782,8.092,149.483
C02472=1110.139,101.009,-58.396,-179.784,8.088,149.482
C02473=1110.144,100.760,-58.377,-179.785,8.084,149.482
C02474=1110.148,100.511,-58.358,-179.787,8.080,149.482
C02475=1110.153,100.262,-58.338,-179.789,8.076,149.481
C02476=1110.158,100.013,-58.319,-179.790,8.073,149.481
C02477=1110.163,99.763,-58.299,-179.792,8.069,149.480
C02478=1110.168,99.515,-58.280,-179.794,8.065,149.480
C02479=1110.172,99.265,-58.261,-179.795,8.061,149.480
C02480=1110.177,99.015,-58.241,-179.797,8.057,149.479
C02481=1110.182,98.767,-58.222,-179.799,8.053,149.479
C02482=1110.187,98.517,-58.203,-179.800,8.050,149.478
C02483=1110.192,98.268,-58.183,-179.801,8.046,149.478
C02484=1110.196,98.019,-58.164,-179.803,8.043,149.477
C02485=1110.201,97.770,-58.145,-179.804,8.039,149.477
C02486=1110.206,97.521,-58.125,-179.806,8.035,149.477
C02487=1110.211,97.272,-58.107,-179.808,8.031,149.476
C02488=1110.216,97.022,-58.088,-179.809,8.027,149.476
C02489=1110.220,96.772,-58.068,-179.811,8.023,149.475
C02490=1110.225,96.524,-58.049,-179.812,8.020,149.475
C02491=1110.230,96.274,-58.030,-179.813,8.016,149.474
C02492=1110.234,96.026,-58.011,-179.815,8.012,149.474
C02493=1110.239,95.776,-57.992,-179.817,8.008,149.473
C02494=1110.245,95.527,-57.973,-179.818,8.004,149.473
C02495=1110.249,95.277,-57.954,-179.820,8.001,149.473
C02496=1110.254,95.029,-57.934,-179.821,7.997,149.472
C02497=1110.258,94.779,-57.916,-179.822,7.994,149.472
C02498=1110.264,94.530,-57.897,-179.824,7.990,149.471
C02499=1110.268,94.281,-57.878,-179.826,7.986,149.471
C02500=1110.273,94.032,-57.858,-179.827,7.982,149.470
C02501=1110.277,93.782,-57.840,-179.828,7.978,149.470
C02502=1110.283,93.533,-57.821,-179.829,7.975,149.469
C02503=1110.287,93.284,-57.802,-179.831,7.971,149.469
C02504=1110.292,93.034,-57.783,-179.833,7.967,149.469
C02505=1110.297,92.786,-57.764,-179.834,7.963,149.468
C02506=1110.302,92.536,-57.745,-179.836,7.959,149.468
C02507=1110.307,92.287,-57.727,-179.836,7.956,149.467
C02508=1110.311,92.072,-57.710,-179.838,7.952,149.467
C02509=1110.315,91.859,-57.693,-179.839,7.949,149.466
C02510=1110.319,91.646,-57.678,-179.840,7.946,149.466
C02511=1110.323,91.432,-57.662,-179.841,7.943,149.465
C02512=1110.327,91.217,-57.645,-179.843,7.939,149.465
C02513=1110.332,91.004,-57.629,-179.844,7.936,149.465
C02514=1110.336,90.790,-57.613,-179.845,7.933,149.464
C02515=1110.340,90.576,-57.597,-179.846,7.929,149.464
C02516=1110.344,90.327,-57.578,-179.847,7.926,149.463
C02517=1110.350,90.077,-57.560,-179.849,7.922,149.463
C02518=1110.354,89.828,-57.541,-179.849,7.918,149.462
C02519=1110.360,89.579,-57.522,-179.851,7.914,149.462
C02520=1110.364,89.329,-57.503,-179.853,7.910,149.461
C02521=1110.368,89.080,-57.485,-179.854,7.906,149.461
C02522=1110.374,88.831,-57.466,-179.855,7.903,149.460
C02523=1110.378,88.582,-57.447,-179.856,7.899,149.460
C02524=1110.383,88.333,-57.429,-179.858,7.895,149.459
C02525=1110.388,88.084,-57.410,-179.858,7.892,149.459
C02526=1110.392,87.834,-57.391,-179.860,7.888,149.458
C02527=1110.398,87.585,-57.372,-179.861,7.884,149.458
C02528=1110.403,87.336,-57.354,-179.863,7.880,149.457
C02529=1110.407,87.086,-57.335,-179.864,7.877,149.457
C02530=1110.412,86.837,-57.316,-179.865,7.872,149.456
C02531=1110.417,86.588,-57.298,-179.866,7.868,149.456
C02532=1110.421,86.338,-57.280,-179.867,7.865,149.455
C02533=1110.427,86.090,-57.260,-179.868,7.861,149.455
C02534=1110.432,85.840,-57.242,-179.870,7.857,149.454
C02535=1110.436,85.590,-57.224,-179.871,7.854,149.454
C02536=1110.441,85.342,-57.205,-179.872,7.850,149.453
C02537=1110.446,85.092,-57.187,-179.874,7.846,149.453
C02538=1110.451,84.843,-57.168,-179.874,7.842,149.452
C02539=1110.455,84.594,-57.150,-179.876,7.838,149.452
C02540=1110.460,84.345,-57.132,-179.876,7.835,149.451
C02541=1110.465,84.095,-57.113,-179.878,7.831,149.451
C02542=1110.470,83.846,-57.094,-179.879,7.827,149.450
C02543=1110.475,83.597,-57.076,-179.880,7.824,149.449
C02544=1110.480,83.348,-57.058,-179.881,7.819,149.449
C02545=1110.484,83.098,-57.039,-179.882,7.816,149.448
C02546=1110.489,82.849,-57.021,-179.883,7.812,149.448
C02547=1110.494,82.600,-57.003,-179.885,7.808,149.447
C02548=1110.498,82.350,-56.984,-179.885,7.805,149.447
C02549=1110.504,82.101,-56.965,-179.887,7.801,149.446
C02550=1110.509,81.852,-56.947,-179.888,7.798,149.446
C02551=1110.514,81.603,-56.929,-179.889,7.793,149.445
C02552=1110.518,81.353,-56.911,-179.890,7.790,149.444
C02553=1110.523,81.104,-56.893,-179.891,7.786,149.444
C02554=1110.527,80.855,-56.874,-179.892,7.782,149.443
C02555=1110.533,80.606,-56.855,-179.893,7.779,149.443
C02556=1110.537,80.356,-56.837,-179.894,7.774,149.442
C02557=1110.542,80.107,-56.819,-179.895,7.771,149.442
C02558=1110.547,79.857,-56.801,-179.896,7.767,149.441
C02559=1110.552,79.608,-56.783,-179.897,7.764,149.441
C02560=1110.557,79.359,-56.765,-179.899,7.759,149.440
C02561=1110.561,79.110,-56.746,-179.900,7.756,149.440
C02562=1110.567,78.860,-56.728,-179.901,7.752,149.439
C02563=1110.572,78.611,-56.710,-179.902,7.749,149.439
C02564=1110.576,78.396,-56.694,-179.902,7.745,149.438
C02565=1110.579,78.183,-56.679,-179.903,7.742,149.438
C02566=1110.584,77.970,-56.663,-179.904,7.739,149.437
C02567=1110.588,77.755,-56.648,-179.905,7.736,149.437
C02568=1110.592,77.542,-56.632,-179.906,7.733,149.436
C02569=1110.596,77.328,-56.616,-179.906,7.730,149.436
C02570=1110.601,77.114,-56.601,-179.907,7.726,149.435
C02571=1110.605,76.900,-56.585,-179.908,7.723,149.435
C02572=1110.610,76.650,-56.567,-179.910,7.719,149.434
C02573=1110.615,76.401,-56.549,-179.911,7.715,149.434
C02574=1110.620,76.152,-56.531,-179.913,7.711,149.433
C02575=1110.624,75.902,-56.513,-179.914,7.707,149.433
C02576=1110.629,75.653,-56.495,-179.915,7.704,149.432
C02577=1110.634,75.404,-56.477,-179.916,7.700,149.432
C02578=1110.639,75.155,-56.459,-179.918,7.696,149.431
C02579=1110.644,74.906,-56.441,-179.919,7.692,149.431
C02580=1110.648,74.656,-56.423,-179.921,7.688,149.430
C02581=1110.654,74.407,-56.405,-179.922,7.684,149.430
C02582=1110.659,74.157,-56.388,-179.924,7.680,149.429
C02583=1110.663,73.907,-56.369,-179.925,7.676,149.429
C02584=1110.668,73.658,-56.351,-179.926,7.672,149.428
C02585=1110.673,73.409,-56.333,-179.928,7.668,149.428
C02586=1110.678,73.160,-56.315,-179.930,7.664,149.427
C02587=1110.683,72.911,-56.297,-179.931,7.660,149.427
C02588=1110.687,72.662,-56.279,-179.932,7.657,149.426
C02589=1110.692,72.412,-56.261,-179.933,7.653,149.426
C02590=1110.698,72.163,-56.244,-179.934,7.648,149.425
C02591=1110.702,71.913,-56.226,-179.936,7.645,149.425
C02592=1110.707,71.665,-56.209,-179.937,7.641,149.424
C02593=1110.712,71.415,-56.191,-179.939,7.637,149.424
C02594=1110.716,71.166,-56.172,-179.940,7.632,149.423
C02595=1110.721,70.916,-56.155,-179.942,7.629,149.423
C02596=1110.726,70.667,-56.137,-179.943,7.625,149.422
C02597=1110.731,70.417,-56.119,-179.944,7.620,149.422
C02598=1110.736,70.168,-56.101,-179.945,7.617,149.421
C02599=1110.741,69.918,-56.084,-179.947,7.613,149.421
C02600=1110.746,69.669,-56.066,-179.948,7.609,149.420
C02601=1110.750,69.420,-56.049,-179.950,7.605,149.420
C02602=1110.755,69.171,-56.031,-179.951,7.601,149.419
C02603=1110.760,68.921,-56.013,-179.952,7.597,149.419
C02604=1110.765,68.672,-55.995,-179.954,7.593,149.418
C02605=1110.770,68.422,-55.978,-179.955,7.589,149.418
C02606=1110.775,68.174,-55.961,-179.956,7.586,149.417
C02607=1110.779,67.924,-55.943,-179.958,7.582,149.417
C02608=1110.785,67.675,-55.925,-179.959,7.578,149.416
C02609=1110.790,67.425,-55.907,-179.960,7.574,149.416
C02610=1110.794,67.176,-55.889,-179.962,7.570,149.415
C02611=1110.799,66.927,-55.873,-179.963,7.565,149.415
C02612=1110.804,66.678,-55.855,-179.964,7.561,149.414
C02613=1110.809,66.428,-55.838,-179.966,7.558,149.414
C02614=1110.814,66.179,-55.820,-179.967,7.554,149.413
C02615=1110.818,65.930,-55.802,-179.968,7.550,149.413
C02616=1110.823,65.680,-55.785,-179.970,7.546,149.412
C02617=1110.828,65.431,-55.767,-179.971,7.542,149.412
C02618=1110.834,65.181,-55.750,-179.972,7.538,149.411
C02619=1110.838,64.932,-55.732,-179.973,7.534,149.410
C02620=1110.842,64.718,-55.717,-179.974,7.531,149.410
C02621=1110.846,64.504,-55.703,-179.975,7.528,149.410
C02622=1110.851,64.290,-55.688,-179.977,7.524,149.409
C02623=1110.855,64.076,-55.672,-179.978,7.521,149.409
C02624=1110.859,63.862,-55.658,-179.979,7.517,149.408
C02625=1110.864,63.648,-55.643,-179.980,7.513,149.408
C02626=1110.867,63.434,-55.628,-179.981,7.510,149.407
C02627=1110.872,63.220,-55.613,-179.982,7.507,149.407
C02628=1110.876,62.971,-55.596,-179.983,7.503,149.406
C02629=1110.882,62.721,-55.579,-179.985,7.499,149.406
C02630=1110.886,62.472,-55.561,-179.986,7.495,149.405
C02631=1110.891,62.223,-55.544,-179.988,7.491,149.405
C02632=1110.896,61.974,-55.526,-179.989,7.487,149.404
C02633=1110.901,61.724,-55.510,-179.990,7.483,149.404
C02634=1110.906,61.474,-55.492,-179.991,7.480,149.403
C02635=1110.911,61.225,-55.474,-179.992,7.475,149.403
C02636=1110.915,60.976,-55.458,-179.994,7.471,149.402
C02637=1110.921,60.726,-55.440,-179.995,7.467,149.402
C02638=1110.925,60.477,-55.423,-179.996,7.463,149.401
C02639=1110.931,60.228,-55.406,-179.997,7.460,149.401
C02640=1110.936,59.978,-55.389,-179.999,7.456,149.400
C02641=1110.940,59.729,-55.371,180.000,7.452,149.400
C02642=1110.945,59.480,-55.354,179.999,7.448,149.399
C02643=1110.950,59.230,-55.338,179.997,7.444,149.399
C02644=1110.955,58.980,-55.320,179.996,7.439,149.398
C02645=1110.960,58.732,-55.303,179.995,7.436,149.397
C02646=1110.965,58.482,-55.286,179.994,7.432,149.397
C02647=1110.969,58.233,-55.269,179.993,7.428,149.396
C02648=1110.975,57.983,-55.252,179.991,7.424,149.396
C02649=1110.979,57.734,-55.235,179.990,7.420,149.395
C02650=1110.985,57.485,-55.218,179.989,7.415,149.395
C02651=1110.989,57.236,-55.201,179.988,7.412,149.394
C02652=1110.994,56.986,-55.184,179.987,7.408,149.394
C02653=1110.999,56.736,-55.167,179.985,7.404,149.393
C02654=1111.004,56.487,-55.149,179.984,7.400,149.392
C02655=1111.009,56.238,-55.133,179.983,7.396,149.392
C02656=1111.014,55.989,-55.116,179.981,7.392,149.391
C02657=1111.019,55.739,-55.099,179.981,7.388,149.391
C02658=1111.024,55.489,-55.082,179.979,7.384,149.390
C02659=1111.029,55.241,-55.065,179.978,7.380,149.390
C02660=1111.034,54.991,-55.048,179.977,7.376,149.389
C02661=1111.039,54.741,-55.031,179.976,7.372,149.389
C02662=1111.043,54.492,-55.014,179.974,7.368,149.388
C02663=1111.049,54.243,-54.997,179.974,7.364,149.387
C02664=1111.053,53.994,-54.981,179.972,7.360,149.387
C02665=1111.058,53.744,-54.963,179.971,7.356,149.386
C02666=1111.063,53.495,-54.947,179.970,7.352,149.386
C02667=1111.068,53.246,-54.930,179.968,7.348,149.385
C02668=1111.073,52.996,-54.913,179.968,7.344,149.385
C02669=1111.078,52.746,-54.896,179.966,7.340,149.384
C02670=1111.083,52.497,-54.879,179.965,7.336,149.384
C02671=1111.088,52.248,-54.863,179.964,7.332,149.383
C02672=1111.092,51.998,-54.846,179.963,7.328,149.382
C02673=1111.098,51.749,-54.829,179.962,7.324,149.382
C02674=1111.103,51.500,-54.813,179.961,7.321,149.381
C02675=1111.107,51.250,-54.796,179.959,7.316,149.381
C02676=1111.112,51.036,-54.782,179.959,7.313,149.380
C02677=1111.116,50.822,-54.767,179.957,7.309,149.380
C02678=1111.120,50.608,-54.753,179.957,7.306,149.379
C02679=1111.124,50.394,-54.739,179.956,7.303,149.379
C02680=1111.129,50.180,-54.724,179.954,7.299,149.378
C02681=1111.133,49.966,-54.710,179.954,7.295,149.378
C02682=1111.137,49.751,-54.695,179.953,7.292,149.377
C02683=1111.141,49.537,-54.682,179.952,7.289,149.377
C02684=1111.146,49.288,-54.665,179.951,7.285,149.376
C02685=1111.151,49.038,-54.648,179.950,7.280,149.376
C02686=1111.156,48.789,-54.632,179.948,7.276,149.375
C02687=1111.161,48.540,-54.615,179.947,7.272,149.374
C02688=1111.165,48.291,-54.599,179.946,7.269,149.374
C02689=1111.172,48.041,-54.582,179.945,7.265,149.373
C02690=1111.176,47.791,-54.566,179.944,7.260,149.373
C02691=1111.181,47.542,-54.549,179.943,7.256,149.372
C02692=1111.186,47.293,-54.533,179.941,7.252,149.372
C02693=1111.190,47.044,-54.516,179.941,7.249,149.371
C02694=1111.196,46.793,-54.500,179.940,7.244,149.370
C02695=1111.201,46.544,-54.483,179.939,7.240,149.370
C02696=1111.205,46.295,-54.467,179.937,7.236,149.369
C02697=1111.210,46.046,-54.450,179.936,7.232,149.369
C02698=1111.215,45.796,-54.434,179.935,7.228,149.368
C02699=1111.220,45.547,-54.418,179.934,7.224,149.367
C02700=1111.225,45.298,-54.401,179.933,7.220,149.367
C02701=1111.230,45.047,-54.385,179.932,7.216,149.366
C02702=1111.235,44.799,-54.368,179.931,7.211,149.366
C02703=1111.240,44.549,-54.352,179.930,7.208,149.365
C02704=1111.245,44.300,-54.336,179.929,7.204,149.364
C02705=1111.250,44.050,-54.320,179.928,7.200,149.364
C02706=1111.255,43.801,-54.303,179.927,7.195,149.363
C02707=1111.260,43.551,-54.287,179.925,7.191,149.363
C02708=1111.265,43.302,-54.270,179.925,7.188,149.362
C02709=1111.270,43.053,-54.254,179.923,7.184,149.361
C02710=1111.274,42.803,-54.238,179.922,7.179,149.361
C02711=1111.280,42.554,-54.221,179.921,7.175,149.360
C02712=1111.284,42.304,-54.206,179.920,7.171,149.359
C02713=1111.289,42.055,-54.189,179.920,7.167,149.359
C02714=1111.294,41.806,-54.173,179.918,7.163,149.358
C02715=1111.299,41.556,-54.157,179.917,7.159,149.358
C02716=1111.304,41.307,-54.140,179.916,7.155,149.357
C02717=1111.309,41.057,-54.125,179.915,7.150,149.356
C02718=1111.314,40.808,-54.108,179.915,7.147,149.356
C02719=1111.319,40.558,-54.092,179.913,7.143,149.355
C02720=1111.324,40.309,-54.076,179.912,7.138,149.354
C02721=1111.329,40.059,-54.060,179.911,7.134,149.354
C02722=1111.334,39.811,-54.044,179.910,7.130,149.353
C02723=1111.339,39.561,-54.028,179.909,7.127,149.353
C02724=1111.344,39.312,-54.012,179.908,7.122,149.352
C02725=1111.349,39.062,-53.996,179.907,7.118,149.351
C02726=1111.354,38.813,-53.979,179.906,7.114,149.351
C02727=1111.358,38.563,-53.963,179.906,7.110,149.350
C02728=1111.364,38.313,-53.948,179.905,7.106,149.349
C02729=1111.368,38.064,-53.931,179.904,7.102,149.349
C02730=1111.374,37.815,-53.916,179.902,7.097,149.348
C02731=1111.379,37.566,-53.899,179.901,7.093,149.347
C02732=1111.383,37.351,-53.886,179.900,7.090,149.347
C02733=1111.387,37.137,-53.872,179.900,7.086,149.346
C02734=1111.392,36.923,-53.858,179.899,7.083,149.346
C02735=1111.396,36.708,-53.844,179.898,7.079,149.345
C02736=1111.400,36.494,-53.831,179.897,7.076,149.345
C02737=1111.405,36.280,-53.817,179.897,7.072,149.344
C02738=1111.409,36.065,-53.803,179.896,7.069,149.344
C02739=1111.413,35.851,-53.790,179.895,7.065,149.343
C02740=1111.418,35.603,-53.774,179.894,7.060,149.342
C02741=1111.422,35.353,-53.758,179.893,7.057,149.342
C02742=1111.428,35.103,-53.742,179.892,7.053,149.341
C02743=1111.433,34.854,-53.727,179.891,7.048,149.341
C02744=1111.438,34.604,-53.710,179.890,7.044,149.340
C02745=1111.443,34.355,-53.695,179.889,7.040,149.339
C02746=1111.448,34.105,-53.679,179.888,7.036,149.339
C02747=1111.453,33.855,-53.663,179.887,7.032,149.338
C02748=1111.457,33.607,-53.647,179.886,7.028,149.337
C02749=1111.463,33.358,-53.632,179.885,7.023,149.337
C02750=1111.468,33.107,-53.616,179.885,7.020,149.336
C02751=1111.473,32.858,-53.600,179.884,7.015,149.335
C02752=1111.478,32.609,-53.583,179.883,7.011,149.334
C02753=1111.482,32.359,-53.568,179.882,7.006,149.334
C02754=1111.488,32.110,-53.553,179.881,7.002,149.333
C02755=1111.493,31.861,-53.537,179.881,6.999,149.332
C02756=1111.498,31.611,-53.521,179.880,6.994,149.332
C02757=1111.503,31.361,-53.506,179.879,6.990,149.331
C02758=1111.507,31.113,-53.490,179.877,6.986,149.330
C02759=1111.512,30.863,-53.474,179.876,6.981,149.330
C02760=1111.518,30.613,-53.458,179.876,6.977,149.329
C02761=1111.523,30.364,-53.443,179.875,6.973,149.328
C02762=1111.527,30.114,-53.428,179.874,6.969,149.328
C02763=1111.532,29.865,-53.412,179.873,6.965,149.327
C02764=1111.538,29.615,-53.396,179.872,6.960,149.326
C02765=1111.543,29.365,-53.380,179.872,6.957,149.326
C02766=1111.547,29.116,-53.365,179.871,6.952,149.325
C02767=1111.553,28.867,-53.350,179.870,6.948,149.324
C02768=1111.558,28.618,-53.334,179.869,6.943,149.323
C02769=1111.562,28.368,-53.318,179.868,6.939,149.323
C02770=1111.567,28.119,-53.303,179.868,6.936,149.322
C02771=1111.573,27.869,-53.287,179.867,6.931,149.321
C02772=1111.577,27.620,-53.272,179.866,6.927,149.321
C02773=1111.582,27.370,-53.256,179.865,6.922,149.320
C02774=1111.587,27.121,-53.240,179.864,6.918,149.319
C02775=1111.592,26.871,-53.225,179.863,6.914,149.319
C02776=1111.597,26.622,-53.210,179.863,6.910,149.318
C02777=1111.602,26.372,-53.194,179.862,6.905,149.317
C02778=1111.607,26.122,-53.180,179.861,6.901,149.316
C02779=1111.613,25.873,-53.164,179.860,6.896,149.316
C02780=1111.618,25.623,-53.148,179.859,6.892,149.315
C02781=1111.623,25.374,-53.133,179.859,6.889,149.314
C02782=1111.627,25.124,-53.118,179.858,6.884,149.314
C02783=1111.632,24.875,-53.103,179.857,6.880,149.313
C02784=1111.637,24.626,-53.087,179.856,6.875,149.312
C02785=1111.643,24.376,-53.071,179.855,6.871,149.311
C02786=1111.647,24.127,-53.056,179.855,6.867,149.311
C02787=1111.652,23.877,-53.040,179.854,6.863,149.310
C02788=1111.657,23.663,-53.028,179.853,6.859,149.309
C02789=1111.661,23.449,-53.015,179.852,6.855,149.309
C02790=1111.666,23.234,-53.002,179.852,6.851,149.308
C02791=1111.669,23.020,-52.989,179.852,6.848,149.307
C02792=1111.674,22.806,-52.975,179.850,6.843,149.307
C02793=1111.678,22.592,-52.963,179.850,6.840,149.306
C02794=1111.682,22.377,-52.949,179.849,6.837,149.306
C02795=1111.687,22.162,-52.936,179.849,6.833,149.305
C02796=1111.691,21.913,-52.921,179.848,6.829,149.304
C02797=1111.697,21.664,-52.906,179.847,6.824,149.303
C02798=1111.701,21.415,-52.891,179.847,6.820,149.302
C02799=1111.707,21.165,-52.876,179.845,6.815,149.302
C02800=1111.712,20.916,-52.861,179.845,6.812,149.301
C02801=1111.717,20.666,-52.845,179.844,6.807,149.300
C02802=1111.721,20.417,-52.830,179.843,6.803,149.300
C02803=1111.727,20.166,-52.815,179.843,6.798,149.299
C02804=1111.732,19.917,-52.800,179.842,6.794,149.298
C02805=1111.737,19.668,-52.784,179.841,6.789,149.297
C02806=1111.742,19.418,-52.770,179.841,6.785,149.296
C02807=1111.747,19.169,-52.755,179.840,6.781,149.296
C02808=1111.752,18.920,-52.739,179.839,6.776,149.295
C02809=1111.757,18.671,-52.724,179.839,6.772,149.294
C02810=1111.762,18.421,-52.710,179.838,6.767,149.293
C02811=1111.767,18.172,-52.695,179.837,6.763,149.293
C02812=1111.772,17.921,-52.679,179.837,6.759,149.292
C02813=1111.777,17.672,-52.664,179.836,6.754,149.291
C02814=1111.781,17.423,-52.649,179.836,6.750,149.290
C02815=1111.787,17.173,-52.634,179.834,6.745,149.289
C02816=1111.792,16.924,-52.619,179.834,6.741,149.289
C02817=1111.797,16.674,-52.604,179.833,6.736,149.288
C02818=1111.802,16.424,-52.590,179.833,6.733,149.287
C02819=1111.807,16.175,-52.575,179.832,6.728,149.286
C02820=1111.812,15.925,-52.560,179.831,6.723,149.286
C02821=1111.817,15.676,-52.545,179.831,6.719,149.285
C02822=1111.822,15.427,-52.530,179.830,6.714,149.284
C02823=1111.827,15.177,-52.515,179.829,6.710,149.283
C02824=1111.832,14.927,-52.501,179.829,6.706,149.282
C02825=1111.837,14.678,-52.486,179.828,6.702,149.282
C02826=1111.843,14.428,-52.471,179.828,6.697,149.281
C02827=1111.847,14.179,-52.456,179.827,6.692,149.280
C02828=1111.852,13.930,-52.441,179.826,6.688,149.279
C02829=1111.858,13.680,-52.426,179.825,6.683,149.278
C02830=1111.863,13.430,-52.412,179.826,6.679,149.277
C02831=1111.867,13.181,-52.397,179.825,6.674,149.276
C02832=1111.873,12.931,-52.382,179.824,6.670,149.276
C02833=1111.878,12.682,-52.367,179.823,6.665,149.275
C02834=1111.883,12.432,-52.352,179.823,6.661,149.274
C02835=1111.887,12.183,-52.338,179.822,6.656,149.273
C02836=1111.893,11.933,-52.323,179.821,6.652,149.272
C02837=1111.898,11.684,-52.308,179.821,6.648,149.272
C02838=1111.903,11.435,-52.293,179.821,6.643,149.271
C02839=1111.907,11.185,-52.279,179.820,6.638,149.270
C02840=1111.913,10.935,-52.263,179.819,6.634,149.269
C02841=1111.918,10.686,-52.249,179.819,6.629,149.268
C02842=1111.923,10.436,-52.235,179.818,6.625,149.267
C02843=1111.927,10.187,-52.220,179.818,6.620,149.267
C02844=1111.933,9.973,-52.207,179.817,6.616,149.266
C02845=1111.936,9.758,-52.195,179.817,6.612,149.265
C02846=1111.940,9.543,-52.183,179.817,6.609,149.264
C02847=1111.946,9.329,-52.170,179.816,6.605,149.264
C02848=1111.949,9.115,-52.158,179.815,6.601,149.263
C02849=1111.954,8.901,-52.145,179.815,6.597,149.262
C02850=1111.958,8.686,-52.132,179.814,6.593,149.261
C02851=1111.963,8.472,-52.120,179.814,6.589,149.261
C02852=1111.968,8.223,-52.105,179.813,6.585,149.260
C02853=1111.973,7.973,-52.091,179.813,6.580,149.259
C02854=1111.977,7.723,-52.077,179.812,6.575,149.258
C02855=1111.983,7.474,-52.061,179.812,6.570,149.257
C02856=1111.988,7.224,-52.047,179.811,6.566,149.256
C02857=1111.993,6.974,-52.033,179.811,6.561,149.255
C02858=1111.998,6.725,-52.018,179.810,6.557,149.255
C02859=1112.003,6.475,-52.004,179.809,6.552,149.254
C02860=1112.008,6.227,-51.990,179.809,6.547,149.253
C02861=1112.013,5.977,-51.975,179.808,6.543,149.252
C02862=1112.018,5.727,-51.961,179.808,6.539,149.251
C02863=1112.023,5.477,-51.947,179.807,6.534,149.251
C02864=1112.028,5.228,-51.932,179.807,6.530,149.250
C02865=1112.033,4.978,-51.918,179.806,6.525,149.249
C02866=1112.038,4.729,-51.903,179.806,6.520,149.248
C02867=1112.044,4.480,-51.889,179.805,6.516,149.247
C02868=1112.049,4.230,-51.874,179.804,6.511,149.246
C02869=1112.054,3.980,-51.860,179.803,6.506,149.246
C02870=1112.059,3.731,-51.846,179.803,6.502,149.245
C02871=1112.063,3.481,-51.832,179.802,6.497,149.244
C02872=1112.068,3.231,-51.817,179.801,6.493,149.243
C02873=1112.074,2.982,-51.803,179.801,6.488,149.242
C02874=1112.079,2.732,-51.789,179.801,6.484,149.241
C02875=1112.084,2.483,-51.775,179.800,6.479,149.240
C02876=1112.089,2.233,-51.761,179.799,6.475,149.240
C02877=1112.093,1.984,-51.746,179.799,6.470,149.239
C02878=1112.099,1.735,-51.732,179.798,6.466,149.238
C02879=1112.104,1.485,-51.717,179.797,6.461,149.237
C02880=1112.109,1.235,-51.703,179.797,6.457,149.236
C02881=1112.114,0.986,-51.689,179.796,6.452,149.236
C02882=1112.119,0.736,-51.675,179.796,6.447,149.235
C02883=1112.124,0.487,-51.661,179.795,6.443,149.234
C02884=1112.129,0.237,-51.646,179.794,6.438,149.233
C02885=1112.135,-0.013,-51.633,179.794,6.434,149.232
C02886=1112.140,-0.263,-51.619,179.794,6.429,149.231
C02887=1112.144,-0.511,-51.605,179.793,6.425,149.231
C02888=1112.149,-0.761,-51.591,179.792,6.420,149.230
C02889=1112.154,-1.011,-51.577,179.792,6.416,149.229
C02890=1112.159,-1.261,-51.562,179.791,6.411,149.228
C02891=1112.165,-1.510,-51.548,179.790,6.407,149.227
C02892=1112.170,-1.759,-51.534,179.790,6.402,149.226
C02893=1112.175,-2.009,-51.520,179.789,6.397,149.226
C02894=1112.180,-2.259,-51.506,179.788,6.393,149.225
C02895=1112.185,-2.508,-51.492,179.788,6.389,149.224
C02896=1112.191,-2.758,-51.478,179.788,6.384,149.223
C02897=1112.195,-3.007,-51.464,179.787,6.380,149.222
C02898=1112.200,-3.256,-51.451,179.786,6.375,149.222
C02899=1112.205,-3.506,-51.436,179.786,6.370,149.221
C02900=1112.210,-3.720,-51.424,179.785,6.367,149.220
C02901=1112.214,-3.935,-51.413,179.784,6.363,149.219
C02902=1112.218,-4.149,-51.401,179.784,6.359,149.219
C02903=1112.223,-4.365,-51.389,179.784,6.355,149.218
C02904=1112.227,-4.578,-51.377,179.783,6.351,149.217
C02905=1112.231,-4.793,-51.364,179.783,6.347,149.216
C02906=1112.236,-5.008,-51.353,179.782,6.344,149.216
C02907=1112.240,-5.222,-51.341,179.781,6.339,149.215
C02908=1112.245,-5.471,-51.327,179.781,6.335,149.214
C02909=1112.250,-5.722,-51.313,179.780,6.330,149.213
C02910=1112.256,-5.971,-51.299,179.780,6.326,149.213
C02911=1112.261,-6.220,-51.285,179.779,6.322,149.212
C02912=1112.265,-6.470,-51.271,179.779,6.317,149.211
C02913=1112.271,-6.719,-51.258,179.778,6.312,149.210
C02914=1112.276,-6.969,-51.244,179.777,6.308,149.209
C02915=1112.281,-7.219,-51.230,179.777,6.303,149.208
C02916=1112.286,-7.468,-51.217,179.776,6.298,149.208
C02917=1112.291,-7.718,-51.203,179.775,6.294,149.207
C02918=1112.296,-7.967,-51.189,179.775,6.289,149.206
C02919=1112.302,-8.217,-51.175,179.774,6.285,149.205
C02920=1112.306,-8.467,-51.162,179.774,6.281,149.204
C02921=1112.311,-8.716,-51.148,179.773,6.276,149.203
C02922=1112.317,-8.966,-51.134,179.773,6.272,149.203
C02923=1112.321,-9.215,-51.120,179.772,6.267,149.202
C02924=1112.327,-9.465,-51.107,179.772,6.262,149.201
C02925=1112.332,-9.715,-51.093,179.771,6.258,149.200
C02926=1112.337,-9.963,-51.080,179.770,6.253,149.199
C02927=1112.342,-10.214,-51.066,179.770,6.248,149.198
C02928=1112.347,-10.463,-51.052,179.769,6.244,149.198
C02929=1112.352,-10.713,-51.039,179.768,6.239,149.197
C02930=1112.357,-10.962,-51.025,179.768,6.235,149.196
C02931=1112.363,-11.212,-51.012,179.768,6.231,149.195
C02932=1112.367,-11.461,-50.998,179.767,6.226,149.194
C02933=1112.372,-11.710,-50.984,179.766,6.222,149.193
C02934=1112.378,-11.961,-50.971,179.766,6.217,149.193
C02935=1112.383,-12.209,-50.957,179.765,6.212,149.192
C02936=1112.388,-12.460,-50.944,179.764,6.208,149.191
C02937=1112.393,-12.709,-50.930,179.764,6.203,149.190
C02938=1112.398,-12.959,-50.917,179.763,6.198,149.189
C02939=1112.403,-13.209,-50.903,179.763,6.194,149.188
C02940=1112.408,-13.458,-50.890,179.762,6.189,149.187
C02941=1112.413,-13.708,-50.876,179.762,6.185,149.187
C02942=1112.418,-13.957,-50.863,179.761,6.181,149.186
C02943=1112.423,-14.207,-50.850,179.761,6.176,149.185
C02944=1112.428,-14.456,-50.836,179.760,6.171,149.184
C02945=1112.433,-14.706,-50.823,179.760,6.167,149.183
C02946=1112.439,-14.956,-50.810,179.759,6.162,149.182
C02947=1112.443,-15.205,-50.796,179.759,6.158,149.182
C02948=1112.449,-15.455,-50.783,179.758,6.153,149.181
C02949=1112.454,-15.704,-50.769,179.758,6.148,149.180
C02950=1112.459,-15.954,-50.756,179.757,6.143,149.179
C02951=1112.464,-16.204,-50.743,179.756,6.139,149.178
C02952=1112.470,-16.453,-50.729,179.756,6.134,149.177
C02953=1112.475,-16.702,-50.716,179.755,6.130,149.176
C02954=1112.480,-16.953,-50.703,179.755,6.125,149.176
C02955=1112.485,-17.201,-50.689,179.755,6.121,149.175
C02956=1112.489,-17.417,-50.678,179.754,6.117,149.174
C02957=1112.494,-17.631,-50.666,179.753,6.113,149.173
C02958=1112.498,-17.845,-50.656,179.753,6.108,149.172
C02959=1112.502,-18.060,-50.644,179.753,6.105,149.172
C02960=1112.507,-18.275,-50.633,179.752,6.101,149.171
C02961=1112.511,-18.489,-50.621,179.752,6.096,149.170
C02962=1112.515,-18.703,-50.610,179.751,6.093,149.169
C02963=1112.520,-18.918,-50.599,179.750,6.089,149.169
C02964=1112.525,-19.168,-50.585,179.750,6.084,149.168
C02965=1112.530,-19.418,-50.572,179.749,6.079,149.167
C02966=1112.535,-19.668,-50.559,179.749,6.074,149.166
C02967=1112.540,-19.917,-50.546,179.748,6.070,149.165
C02968=1112.545,-20.166,-50.533,179.748,6.065,149.164
C02969=1112.551,-20.416,-50.519,179.748,6.061,149.163
C02970=1112.556,-20.666,-50.507,179.748,6.056,149.163
C02971=1112.560,-20.916,-50.494,179.747,6.052,149.162
C02972=1112.566,-21.165,-50.480,179.747,6.047,149.161
C02973=1112.571,-21.414,-50.467,179.746,6.042,149.160
C02974=1112.576,-21.664,-50.454,179.746,6.037,149.159
C02975=1112.581,-21.914,-50.441,179.745,6.033,149.158
C02976=1112.587,-22.163,-50.429,179.745,6.028,149.157
C02977=1112.592,-22.413,-50.415,179.744,6.023,149.156
C02978=1112.597,-22.663,-50.402,179.744,6.018,149.155
C02979=1112.602,-22.912,-50.390,179.743,6.014,149.154
C02980=1112.607,-23.162,-50.375,179.743,6.009,149.154
C02981=1112.612,-23.411,-50.363,179.742,6.004,149.153
C02982=1112.617,-23.660,-50.350,179.742,5.999,149.152
C02983=1112.623,-23.911,-50.337,179.741,5.995,149.151
C02984=1112.628,-24.160,-50.324,179.741,5.990,149.150
C02985=1112.633,-24.409,-50.311,179.740,5.985,149.149
C02986=1112.638,-24.659,-50.298,179.740,5.981,149.148
C02987=1112.643,-24.909,-50.285,179.739,5.976,149.147
C02988=1112.648,-25.158,-50.273,179.739,5.971,149.146
C02989=1112.653,-25.408,-50.260,179.738,5.966,149.145
C02990=1112.659,-25.658,-50.247,179.737,5.961,149.145
C02991=1112.664,-25.907,-50.234,179.738,5.957,149.143
C02992=1112.668,-26.157,-50.221,179.738,5.953,149.143
C02993=1112.673,-26.406,-50.208,179.738,5.947,149.141
C02994=1112.679,-26.656,-50.195,179.738,5.944,149.140
C02995=1112.684,-26.906,-50.182,179.739,5.939,149.139
C02996=1112.689,-27.155,-50.170,179.739,5.935,149.138
C02997=1112.694,-27.405,-50.157,179.739,5.930,149.137
C02998=1112.699,-27.654,-50.144,179.739,5.926,149.136
C02999=1112.705,-27.905,-50.132,179.740,5.922,149.135
C03000=1112.710,-28.154,-50.119,179.739,5.917,149.134
C03001=1112.715,-28.404,-50.106,179.739,5.913,149.133
C03002=1112.720,-28.653,-50.094,179.740,5.909,149.133
C03003=1112.725,-28.903,-50.081,179.740,5.904,149.131
C03004=1112.731,-29.153,-50.068,179.740,5.900,149.131
C03005=1112.736,-29.402,-50.055,179.739,5.895,149.130
C03006=1112.741,-29.651,-50.042,179.739,5.892,149.129
C03007=1112.745,-29.901,-50.029,179.739,5.887,149.128
C03008=1112.750,-30.151,-50.017,179.740,5.883,149.127
C03009=1112.756,-30.400,-50.005,179.739,5.878,149.126
C03010=1112.762,-30.650,-49.992,179.739,5.874,149.125
C03011=1112.766,-30.900,-49.979,179.739,5.869,149.124
C03012=1112.770,-31.114,-49.968,179.738,5.866,149.123
C03013=1112.775,-31.329,-49.957,179.739,5.862,149.122
C03014=1112.779,-31.544,-49.947,179.738,5.858,149.122
C03015=1112.784,-31.758,-49.935,179.738,5.854,149.121
C03016=1112.788,-31.973,-49.925,179.738,5.851,149.120
C03017=1112.793,-32.188,-49.914,179.738,5.847,149.119
C03018=1112.797,-32.402,-49.903,179.738,5.843,149.118
C03019=1112.802,-32.617,-49.892,179.738,5.840,149.118
C03020=1112.807,-32.867,-49.879,179.737,5.835,149.117
C03021=1112.812,-33.117,-49.867,179.737,5.831,149.116
C03022=1112.817,-33.366,-49.855,179.737,5.826,149.115
C03023=1112.822,-33.615,-49.842,179.736,5.821,149.114
C03024=1112.827,-33.864,-49.829,179.735,5.817,149.114
C03025=1112.832,-34.115,-49.817,179.735,5.813,149.113
C03026=1112.837,-34.364,-49.805,179.735,5.808,149.112
C03027=1112.842,-34.614,-49.792,179.735,5.804,149.111
C03028=1112.848,-34.864,-49.780,179.734,5.799,149.110
C03029=1112.853,-35.113,-49.768,179.734,5.794,149.109
C03030=1112.859,-35.363,-49.754,179.733,5.790,149.108
C03031=1112.863,-35.613,-49.741,179.733,5.786,149.107
C03032=1112.869,-35.863,-49.729,179.732,5.781,149.106
C03033=1112.874,-36.112,-49.717,179.732,5.776,149.106
C03034=1112.879,-36.361,-49.704,179.732,5.772,149.105
C03035=1112.884,-36.611,-49.692,179.731,5.767,149.104
C03036=1112.890,-36.860,-49.680,179.730,5.763,149.103
C03037=1112.895,-37.110,-49.668,179.730,5.758,149.102
C03038=1112.900,-37.360,-49.655,179.729,5.753,149.101
C03039=1112.905,-37.610,-49.642,179.728,5.749,149.101
C03040=1112.910,-37.860,-49.630,179.727,5.743,149.100
C03041=1112.915,-38.109,-49.618,179.727,5.738,149.099
C03042=1112.921,-38.359,-49.606,179.726,5.734,149.098
C03043=1112.926,-38.608,-49.593,179.726,5.729,149.097
C03044=1112.931,-38.858,-49.581,179.725,5.725,149.096
C03045=1112.936,-39.107,-49.569,179.724,5.719,149.095
C03046=1112.941,-39.356,-49.557,179.724,5.714,149.094
C03047=1112.946,-39.606,-49.545,179.723,5.710,149.094
C03048=1112.951,-39.856,-49.532,179.723,5.705,149.093
C03049=1112.956,-40.106,-49.520,179.721,5.700,149.092
C03050=1112.961,-40.356,-49.508,179.721,5.695,149.091
C03051=1112.967,-40.606,-49.496,179.720,5.689,149.090
C03052=1112.972,-40.856,-49.484,179.719,5.685,149.089
C03053=1112.977,-41.105,-49.471,179.718,5.679,149.088
C03054=1112.983,-41.355,-49.459,179.718,5.674,149.087
C03055=1112.988,-41.604,-49.447,179.716,5.669,149.087
C03056=1112.992,-41.854,-49.435,179.716,5.664,149.086
C03057=1112.998,-42.103,-49.423,179.715,5.659,149.085
C03058=1113.003,-42.353,-49.411,179.714,5.654,149.084
C03059=1113.008,-42.603,-49.399,179.713,5.649,149.083
C03060=1113.014,-42.852,-49.386,179.712,5.643,149.082
C03061=1113.019,-43.102,-49.375,179.712,5.638,149.081
C03062=1113.023,-43.351,-49.363,179.713,5.634,149.080
C03063=1113.029,-43.601,-49.351,179.713,5.629,149.079
C03064=1113.034,-43.851,-49.339,179.713,5.625,149.078
C03065=1113.039,-44.100,-49.326,179.713,5.619,149.077
C03066=1113.045,-44.350,-49.314,179.713,5.614,149.076
C03067=1113.050,-44.600,-49.303,179.713,5.610,149.075
C03068=1113.055,-44.815,-49.292,179.714,5.606,149.074
C03069=1113.059,-45.029,-49.282,179.714,5.602,149.073
C03070=1113.063,-45.244,-49.272,179.713,5.598,149.072
C03071=1113.067,-45.459,-49.262,179.714,5.593,149.071
C03072=1113.072,-45.674,-49.252,179.714,5.589,149.070
C03073=1113.077,-45.888,-49.241,179.714,5.586,149.069
C03074=1113.081,-46.103,-49.231,179.715,5.582,149.068
C03075=1113.086,-46.318,-49.221,179.715,5.578,149.067
C03076=1113.091,-46.568,-49.209,179.715,5.572,149.066
C03077=1113.095,-46.817,-49.197,179.715,5.569,149.065
C03078=1113.101,-47.066,-49.185,179.715,5.563,149.064
C03079=1113.106,-47.316,-49.173,179.715,5.558,149.063
C03080=1113.112,-47.566,-49.161,179.715,5.554,149.062
C03081=1113.116,-47.815,-49.149,179.715,5.549,149.061
C03082=1113.122,-48.065,-49.137,179.716,5.545,149.060
C03083=1113.127,-48.315,-49.125,179.716,5.540,149.058
C03084=1113.132,-48.565,-49.114,179.716,5.535,149.058
C03085=1113.137,-48.815,-49.102,179.716,5.531,149.056
C03086=1113.142,-49.064,-49.090,179.716,5.526,149.055
C03087=1113.148,-49.313,-49.078,179.717,5.522,149.054
C03088=1113.153,-49.563,-49.067,179.717,5.516,149.053
C03089=1113.158,-49.813,-49.055,179.717,5.511,149.052
C03090=1113.164,-50.063,-49.043,179.717,5.507,149.051
C03091=1113.169,-50.312,-49.032,179.717,5.502,149.050
C03092=1113.174,-50.562,-49.019,179.717,5.497,149.049
C03093=1113.179,-50.812,-49.007,179.717,5.493,149.048
C03094=1113.184,-51.061,-48.996,179.717,5.488,149.047
C03095=1113.189,-51.311,-48.984,179.718,5.484,149.046
C03096=1113.195,-51.561,-48.972,179.718,5.479,149.044
C03097=1113.200,-51.810,-48.961,179.718,5.474,149.043
C03098=1113.205,-52.060,-48.949,179.718,5.470,149.042
C03099=1113.210,-52.310,-48.938,179.718,5.464,149.041
C03100=1113.215,-52.560,-48.926,179.719,5.460,149.040
C03101=1113.221,-52.809,-48.914,179.719,5.455,149.039
C03102=1113.225,-53.059,-48.902,179.719,5.450,149.038
C03103=1113.231,-53.309,-48.890,179.719,5.446,149.037
C03104=1113.236,-53.557,-48.879,179.719,5.441,149.036
C03105=1113.241,-53.807,-48.868,179.719,5.436,149.035
C03106=1113.247,-54.057,-48.856,179.719,5.432,149.034
C03107=1113.252,-54.307,-48.844,179.719,5.427,149.033
C03108=1113.257,-54.557,-48.833,179.720,5.423,149.032
C03109=1113.262,-54.806,-48.821,179.720,5.418,149.031
C03110=1113.268,-55.056,-48.810,179.720,5.413,149.029
C03111=1113.272,-55.305,-48.798,179.720,5.409,149.029
C03112=1113.278,-55.555,-48.787,179.720,5.404,149.027
C03113=1113.283,-55.805,-48.775,179.721,5.399,149.026
C03114=1113.288,-56.055,-48.763,179.720,5.394,149.025
C03115=1113.293,-56.304,-48.752,179.720,5.389,149.024
C03116=1113.299,-56.554,-48.741,179.721,5.385,149.023
C03117=1113.303,-56.803,-48.729,179.721,5.380,149.022
C03118=1113.309,-57.053,-48.717,179.721,5.375,149.021
C03119=1113.314,-57.303,-48.706,179.722,5.371,149.020
C03120=1113.319,-57.553,-48.695,179.721,5.366,149.019
C03121=1113.324,-57.803,-48.684,179.722,5.362,149.018
C03122=1113.330,-58.052,-48.672,179.721,5.357,149.017
C03123=1113.335,-58.302,-48.661,179.722,5.352,149.016
C03124=1113.339,-58.517,-48.651,179.722,5.348,149.015
C03125=1113.343,-58.732,-48.641,179.722,5.344,149.014
C03126=1113.348,-58.947,-48.631,179.722,5.340,149.013
C03127=1113.353,-59.161,-48.621,179.722,5.336,149.012
C03128=1113.357,-59.376,-48.611,179.723,5.332,149.011
C03129=1113.362,-59.591,-48.602,179.723,5.328,149.010
C03130=1113.366,-59.806,-48.592,179.723,5.324,149.009
C03131=1113.371,-60.020,-48.582,179.723,5.319,149.008
C03132=1113.376,-60.270,-48.570,179.722,5.315,149.007
C03133=1113.381,-60.520,-48.559,179.722,5.310,149.006
C03134=1113.386,-60.769,-48.548,179.721,5.304,149.005
C03135=1113.391,-61.020,-48.537,179.720,5.300,149.005
C03136=1113.397,-61.269,-48.526,179.720,5.295,149.004
C03137=1113.402,-61.519,-48.514,179.720,5.290,149.002
C03138=1113.407,-61.768,-48.502,179.719,5.284,149.002
C03139=1113.412,-62.017,-48.492,179.719,5.279,149.001
C03140=1113.418,-62.268,-48.480,179.718,5.275,149.000
C03141=1113.423,-62.517,-48.469,179.718,5.269,148.999
C03142=1113.428,-62.767,-48.457,179.717,5.264,148.998
C03143=1113.433,-63.016,-48.446,179.717,5.259,148.997
C03144=1113.438,-63.267,-48.436,179.717,5.253,148.996
C03145=1113.444,-63.516,-48.424,179.716,5.249,148.995
C03146=1113.449,-63.765,-48.413,179.716,5.244,148.994
C03147=1113.454,-64.016,-48.402,179.716,5.239,148.993
C03148=1113.459,-64.266,-48.390,179.715,5.233,148.992
C03149=1113.465,-64.514,-48.380,179.715,5.228,148.991
C03150=1113.470,-64.765,-48.369,179.715,5.223,148.990
C03151=1113.475,-65.015,-48.357,179.714,5.218,148.989
C03152=1113.480,-65.264,-48.346,179.714,5.212,148.987
C03153=1113.485,-65.514,-48.336,179.713,5.208,148.986
C03154=1113.490,-65.763,-48.324,179.714,5.203,148.985
C03155=1113.496,-66.013,-48.313,179.713,5.197,148.984
C03156=1113.501,-66.263,-48.302,179.713,5.192,148.983
C03157=1113.506,-66.513,-48.291,179.712,5.187,148.982
C03158=1113.511,-66.762,-48.281,179.712,5.182,148.981
C03159=1113.517,-67.012,-48.269,179.711,5.176,148.980
C03160=1113.525,-67.413,-48.252,179.711,5.169,148.979
C03161=1113.534,-67.815,-48.234,179.711,5.160,148.977
C03162=1113.542,-68.217,-48.216,179.711,5.152,148.975
C03163=1113.551,-68.618,-48.198,179.710,5.143,148.973
C03164=1113.556,-68.867,-48.187,179.710,5.138,148.972
C03165=1113.561,-69.118,-48.177,179.710,5.133,148.971
C03166=1113.566,-69.367,-48.166,179.710,5.128,148.970
C03167=1113.572,-69.617,-48.155,179.709,5.123,148.969
C03168=1113.577,-69.867,-48.144,179.710,5.117,148.968
C03169=1113.582,-70.116,-48.133,179.710,5.112,148.967
C03170=1113.587,-70.367,-48.123,179.709,5.107,148.966
C03171=1113.592,-70.615,-48.112,179.709,5.102,148.965
C03172=1113.597,-70.866,-48.101,179.710,5.097,148.964
C03173=1113.603,-71.116,-48.089,179.709,5.091,148.962
C03174=1113.608,-71.365,-48.079,179.709,5.086,148.961
C03175=1113.613,-71.615,-48.068,179.709,5.081,148.960
C03176=1113.619,-71.864,-48.058,179.709,5.076,148.959
C03177=1113.624,-72.115,-48.047,179.709,5.071,148.958
C03178=1113.629,-72.364,-48.036,179.709,5.066,148.957
C03179=1113.634,-72.614,-48.026,179.708,5.060,148.956
C03180=1113.641,-72.892,-48.014,179.709,5.055,148.954
C03181=1113.646,-73.169,-48.001,179.709,5.049,148.953
C03182=1113.652,-73.448,-47.990,179.709,5.044,148.952
C03183=1113.658,-73.725,-47.977,179.709,5.037,148.951
C03184=1113.663,-73.975,-47.967,179.709,5.032,148.950
C03185=1113.669,-74.224,-47.957,179.709,5.027,148.949
C03186=1113.674,-74.475,-47.946,179.709,5.022,148.947
C03187=1113.679,-74.724,-47.935,179.709,5.017,148.946
C03188=1113.684,-74.974,-47.925,179.709,5.012,148.945
C03189=1113.689,-75.223,-47.914,179.709,5.006,148.944
C03190=1113.694,-75.473,-47.903,179.709,5.001,148.943
C03191=1113.700,-75.723,-47.893,179.709,4.996,148.942
C03192=1113.705,-75.973,-47.882,179.709,4.991,148.940
C03193=1113.711,-76.223,-47.872,179.709,4.985,148.939
C03194=1113.716,-76.472,-47.861,179.709,4.980,148.938
C03195=1113.721,-76.722,-47.850,179.709,4.975,148.937
C03196=1113.727,-76.971,-47.840,179.710,4.970,148.936
C03197=1113.732,-77.222,-47.829,179.710,4.965,148.935
C03198=1113.738,-77.471,-47.819,179.710,4.960,148.933
C03199=1113.742,-77.721,-47.808,179.710,4.955,148.932
C03200=1113.748,-77.970,-47.798,179.710,4.949,148.931
C03201=1113.753,-78.220,-47.787,179.710,4.945,148.930
C03202=1113.758,-78.470,-47.777,179.710,4.939,148.929
C03203=1113.764,-78.720,-47.767,179.711,4.934,148.928
C03204=1113.768,-78.970,-47.757,179.711,4.929,148.926
C03205=1113.774,-79.219,-47.746,179.711,4.924,148.925
C03206=1113.779,-79.468,-47.735,179.711,4.919,148.924
C03207=1113.784,-79.718,-47.725,179.711,4.913,148.923
C03208=1113.790,-79.968,-47.715,179.711,4.908,148.922
C03209=1113.795,-80.218,-47.704,179.712,4.903,148.921
C03210=1113.800,-80.468,-47.694,179.712,4.898,148.919
C03211=1113.806,-80.717,-47.684,179.712,4.893,148.918
C03212=1113.811,-80.967,-47.673,179.712,4.888,148.917
C03213=1113.817,-81.217,-47.663,179.712,4.882,148.916
C03214=1113.822,-81.467,-47.652,179.712,4.877,148.915
C03215=1113.827,-81.717,-47.642,179.713,4.872,148.913
C03216=1113.832,-81.965,-47.632,179.713,4.867,148.912
C03217=1113.837,-82.216,-47.621,179.713,4.862,148.911
C03218=1113.842,-82.465,-47.611,179.714,4.858,148.910
C03219=1113.848,-82.715,-47.601,179.714,4.852,148.909
C03220=1113.853,-82.965,-47.590,179.715,4.847,148.907
C03221=1113.859,-83.214,-47.580,179.715,4.842,148.906
C03222=1113.864,-83.464,-47.570,179.715,4.837,148.905
C03223=1113.869,-83.714,-47.559,179.715,4.831,148.904
C03224=1113.874,-83.964,-47.550,179.715,4.826,148.903
C03225=1113.880,-84.213,-47.539,179.716,4.822,148.901
C03226=1113.885,-84.463,-47.529,179.716,4.817,148.900
C03227=1113.890,-84.713,-47.519,179.716,4.812,148.899
C03228=1113.896,-84.962,-47.508,179.717,4.806,148.898
C03229=1113.900,-85.213,-47.499,179.717,4.801,148.897
C03230=1113.906,-85.462,-47.489,179.717,4.796,148.895
C03231=1113.912,-85.712,-47.479,179.718,4.791,148.894
C03232=1113.915,-85.927,-47.470,179.718,4.787,148.893
C03233=1113.921,-86.142,-47.461,179.719,4.782,148.892
C03234=1113.925,-86.357,-47.452,179.719,4.778,148.891
C03235=1113.930,-86.572,-47.443,179.720,4.774,148.890
C03236=1113.934,-86.787,-47.435,179.719,4.769,148.889
C03237=1113.939,-87.002,-47.426,179.720,4.765,148.888
C03238=1113.943,-87.217,-47.417,179.720,4.761,148.887
C03239=1113.947,-87.432,-47.409,179.721,4.757,148.886
C03240=1113.953,-87.681,-47.399,179.721,4.752,148.885
C03241=1113.958,-87.931,-47.388,179.721,4.746,148.883
C03242=1113.964,-88.181,-47.378,179.722,4.741,148.882
C03243=1113.969,-88.431,-47.369,179.722,4.737,148.881
C03244=1113.974,-88.681,-47.358,179.723,4.732,148.880
C03245=1113.979,-88.931,-47.348,179.723,4.726,148.879
C03246=1113.984,-89.180,-47.339,179.724,4.722,148.877
C03247=1113.990,-89.429,-47.328,179.724,4.717,148.876
C03248=1113.995,-89.680,-47.318,179.724,4.711,148.875
C03249=1114.001,-89.930,-47.308,179.725,4.707,148.874
C03250=1114.006,-90.179,-47.299,179.725,4.702,148.872
C03251=1114.011,-90.428,-47.288,179.726,4.697,148.871
C03252=1114.016,-90.679,-47.278,179.726,4.692,148.870
C03253=1114.021,-90.928,-47.268,179.727,4.687,148.869
C03254=1114.027,-91.178,-47.259,179.727,4.683,148.868
C03255=1114.033,-91.428,-47.249,179.728,4.677,148.866
C03256=1114.037,-91.678,-47.239,179.728,4.672,148.865
C03257=1114.042,-91.927,-47.228,179.729,4.668,148.864
C03258=1114.048,-92.177,-47.219,179.729,4.663,148.863
C03259=1114.053,-92.427,-47.209,179.730,4.658,148.861
C03260=1114.059,-92.676,-47.199,179.730,4.653,148.860
C03261=1114.064,-92.926,-47.188,179.731,4.649,148.859
C03262=1114.069,-93.176,-47.180,179.732,4.643,148.858
C03263=1114.075,-93.426,-47.169,179.733,4.639,148.856
C03264=1114.080,-93.675,-47.159,179.733,4.634,148.855
C03265=1114.085,-93.925,-47.150,179.734,4.630,148.854
C03266=1114.090,-94.175,-47.140,179.734,4.624,148.853
C03267=1114.095,-94.425,-47.130,179.734,4.619,148.852
C03268=1114.101,-94.675,-47.121,179.735,4.615,148.851
C03269=1114.107,-94.924,-47.110,179.735,4.610,148.849
C03270=1114.111,-95.174,-47.101,179.735,4.605,148.848
C03271=1114.117,-95.424,-47.091,179.736,4.600,148.847
C03272=1114.122,-95.674,-47.081,179.736,4.595,148.846
C03273=1114.127,-95.923,-47.071,179.736,4.590,148.845
C03274=1114.133,-96.173,-47.062,179.737,4.585,148.843
C03275=1114.138,-96.423,-47.052,179.737,4.580,148.842
C03276=1114.144,-96.672,-47.042,179.738,4.575,148.841
C03277=1114.149,-96.922,-47.033,179.738,4.570,148.840
C03278=1114.154,-97.172,-47.022,179.738,4.565,148.839
C03279=1114.160,-97.422,-47.013,179.739,4.561,148.837
C03280=1114.165,-97.672,-47.003,179.739,4.555,148.836
C03281=1114.170,-97.921,-46.993,179.739,4.550,148.835
C03282=1114.175,-98.171,-46.984,179.740,4.546,148.834
C03283=1114.181,-98.421,-46.974,179.740,4.541,148.833
C03284=1114.186,-98.670,-46.965,179.740,4.536,148.832
C03285=1114.191,-98.921,-46.954,179.740,4.531,148.831
C03286=1114.196,-99.170,-46.946,179.740,4.526,148.829
C03287=1114.202,-99.420,-46.935,179.741,4.521,148.828
C03288=1114.206,-99.634,-46.927,179.741,4.516,148.827
C03289=1114.211,-99.850,-46.919,179.742,4.512,148.826
C03290=1114.215,-100.065,-46.911,179.742,4.508,148.825
C03291=1114.221,-100.280,-46.902,179.743,4.504,148.824
C03292=1114.225,-100.495,-46.894,179.742,4.499,148.823
C03293=1114.229,-100.710,-46.886,179.743,4.495,148.822
C03294=1114.234,-100.925,-46.878,179.743,4.491,148.821
C03295=1114.239,-101.140,-46.870,179.744,4.487,148.820
C03296=1114.244,-101.390,-46.860,179.744,4.482,148.819
C03297=1114.249,-101.640,-46.851,179.744,4.477,148.817
C03298=1114.254,-101.890,-46.841,179.745,4.471,148.816
C03299=1114.260,-102.139,-46.832,179.745,4.467,148.815
C03300=1114.265,-102.389,-46.821,179.746,4.462,148.814
C03301=1114.270,-102.639,-46.813,179.746,4.457,148.813
C03302=1114.276,-102.888,-46.802,179.746,4.452,148.811
C03303=1114.281,-103.138,-46.793,179.746,4.447,148.810
C03304=1114.286,-103.388,-46.785,179.747,4.442,148.809
C03305=1114.292,-103.638,-46.774,179.747,4.437,148.808
C03306=1114.297,-103.888,-46.765,179.747,4.432,148.807
C03307=1114.303,-104.137,-46.755,179.747,4.427,148.806
C03308=1114.308,-104.387,-46.746,179.748,4.422,148.805
C03309=1114.313,-104.637,-46.737,179.748,4.417,148.803
C03310=1114.319,-104.886,-46.727,179.749,4.412,148.802
C03311=1114.323,-105.137,-46.718,179.749,4.407,148.801
C03312=1114.329,-105.386,-46.708,179.749,4.402,148.800
C03313=1114.334,-105.636,-46.699,179.749,4.397,148.799
C03314=1114.339,-105.886,-46.690,179.750,4.392,148.797
C03315=1114.345,-106.136,-46.680,179.750,4.386,148.796
C03316=1114.350,-106.386,-46.671,179.751,4.382,148.795
C03317=1114.355,-106.635,-46.662,179.751,4.377,148.794
C03318=1114.361,-106.885,-46.652,179.751,4.372,148.793
C03319=1114.366,-107.135,-46.643,179.751,4.367,148.791
C03320=1114.371,-107.385,-46.634,179.752,4.361,148.790
C03321=1114.377,-107.635,-46.624,179.752,4.356,148.789
C03322=1114.382,-107.884,-46.615,179.753,4.351,148.787
C03323=1114.387,-108.134,-46.606,179.753,4.346,148.786
C03324=1114.393,-108.384,-46.596,179.754,4.341,148.785
C03325=1114.398,-108.634,-46.588,179.754,4.336,148.784
C03326=1114.403,-108.883,-46.578,179.754,4.331,148.783
C03327=1114.409,-109.133,-46.568,179.754,4.326,148.781
C03328=1114.414,-109.382,-46.560,179.755,4.321,148.780
C03329=1114.420,-109.632,-46.551,179.755,4.315,148.779
C03330=1114.424,-109.881,-46.541,179.755,4.310,148.778
C03331=1114.430,-110.132,-46.532,179.755,4.305,148.777
C03332=1114.436,-110.381,-46.523,179.756,4.300,148.775
C03333=1114.441,-110.631,-46.514,179.756,4.296,148.774
C03334=1114.446,-110.881,-46.505,179.757,4.290,148.773
C03335=1114.452,-111.131,-46.495,179.757,4.285,148.772
C03336=1114.457,-111.381,-46.486,179.757,4.280,148.771
C03337=1114.462,-111.630,-46.477,179.757,4.275,148.769
C03338=1114.467,-111.880,-46.468,179.758,4.270,148.768
C03339=1114.473,-112.130,-46.459,179.758,4.265,148.767
C03340=1114.478,-112.380,-46.450,179.758,4.259,148.766
C03341=1114.483,-112.630,-46.440,179.758,4.254,148.765
C03342=1114.488,-112.879,-46.431,179.759,4.249,148.763
C03343=1114.495,-113.129,-46.422,179.760,4.244,148.762
C03344=1114.498,-113.344,-46.415,179.760,4.240,148.761
C03345=1114.503,-113.559,-46.407,179.760,4.235,148.760
C03346=1114.508,-113.775,-46.400,179.760,4.231,148.759
C03347=1114.513,-113.990,-46.392,179.761,4.227,148.758
C03348=1114.516,-114.205,-46.383,179.761,4.221,148.757
C03349=1114.521,-114.420,-46.376,179.761,4.217,148.756
C03350=1114.526,-114.635,-46.368,179.761,4.213,148.755
C03351=1114.531,-114.850,-46.361,179.762,4.208,148.754
C03352=1114.536,-115.100,-46.352,179.762,4.203,148.752
C03353=1114.541,-115.350,-46.343,179.762,4.198,148.751
C03354=1114.547,-115.600,-46.333,179.763,4.193,148.750
C03355=1114.552,-115.850,-46.324,179.763,4.188,148.749
C03356=1114.558,-116.099,-46.316,179.763,4.182,148.747
C03357=1114.563,-116.349,-46.307,179.764,4.177,148.746
C03358=1114.568,-116.599,-46.298,179.764,4.172,148.745
C03359=1114.574,-116.848,-46.289,179.765,4.167,148.744
C03360=1114.579,-117.098,-46.280,179.765,4.161,148.742
C03361=1114.585,-117.349,-46.271,179.765,4.156,148.741
C03362=1114.590,-117.598,-46.262,179.765,4.151,148.740
C03363=1114.596,-117.848,-46.253,179.766,4.146,148.739
C03364=1114.601,-118.097,-46.244,179.766,4.140,148.737
C03365=1114.606,-118.347,-46.235,179.767,4.135,148.736
C03366=1114.611,-118.597,-46.227,179.767,4.130,148.735
C03367=1114.616,-118.847,-46.218,179.767,4.125,148.734
C03368=1114.622,-119.096,-46.209,179.768,4.120,148.732
C03369=1114.627,-119.346,-46.200,179.768,4.115,148.731
C03370=1114.632,-119.596,-46.191,179.769,4.109,148.730
C03371=1114.638,-119.846,-46.183,179.768,4.103,148.729
C03372=1114.643,-120.096,-46.174,179.769,4.098,148.727
C03373=1114.649,-120.345,-46.166,179.769,4.093,148.726
C03374=1114.655,-120.595,-46.156,179.769,4.087,148.725
C03375=1114.660,-120.845,-46.147,179.770,4.082,148.724
C03376=1114.665,-121.095,-46.138,179.770,4.077,148.722
C03377=1114.670,-121.345,-46.130,179.771,4.072,148.721
C03378=1114.676,-121.594,-46.121,179.771,4.066,148.720
C03379=1114.681,-121.845,-46.113,179.772,4.061,148.718
C03380=1114.687,-122.094,-46.104,179.772,4.056,148.717
C03381=1114.692,-122.344,-46.095,179.772,4.051,148.716
C03382=1114.697,-122.593,-46.087,179.772,4.045,148.715
C03383=1114.703,-122.843,-46.078,179.773,4.039,148.713
C03384=1114.708,-123.094,-46.069,179.773,4.034,148.712
C03385=1114.713,-123.343,-46.061,179.773,4.029,148.711
C03386=1114.718,-123.592,-46.053,179.774,4.024,148.710
C03387=1114.723,-123.842,-46.044,179.774,4.018,148.708
C03388=1114.729,-124.092,-46.035,179.775,4.013,148.707
C03389=1114.734,-124.343,-46.027,179.774,4.007,148.706
C03390=1114.740,-124.592,-46.018,179.775,4.001,148.704
C03391=1114.745,-124.842,-46.009,179.776,3.996,148.703
C03392=1114.751,-125.092,-46.001,179.776,3.991,148.702
C03393=1114.756,-125.341,-45.992,179.776,3.986,148.701
C03394=1114.761,-125.591,-45.984,179.777,3.980,148.699
C03395=1114.767,-125.841,-45.975,179.777,3.974,148.698
C03396=1114.773,-126.091,-45.967,179.777,3.969,148.697
C03397=1114.778,-126.341,-45.958,179.778,3.963,148.695
C03398=1114.783,-126.590,-45.949,179.778,3.958,148.694
C03399=1114.788,-126.841,-45.941,179.778,3.953,148.693
C03400=1114.793,-127.056,-45.934,179.779,3.948,148.692
C03401=1114.797,-127.271,-45.926,179.779,3.943,148.690
C03402=1114.802,-127.486,-45.919,179.779,3.939,148.689
C03403=1114.807,-127.701,-45.912,179.780,3.934,148.688
C03404=1114.811,-127.916,-45.905,179.781,3.929,148.687
C03405=1114.816,-128.131,-45.897,179.780,3.925,148.686
C03406=1114.821,-128.347,-45.891,179.781,3.919,148.685
C03407=1114.825,-128.562,-45.883,179.782,3.915,148.684
C03408=1114.402,-128.552,-45.909,179.788,3.919,148.682
C03409=1114.398,-128.337,-45.916,179.788,3.924,148.684
C03410=1114.393,-128.122,-45.924,179.788,3.929,148.685
C03411=1114.388,-127.906,-45.930,179.787,3.933,148.686
C03412=1114.384,-127.691,-45.938,179.787,3.938,148.687
C03413=1114.379,-127.476,-45.946,179.787,3.942,148.688
C03414=1114.375,-127.262,-45.953,179.786,3.947,148.689
C03415=1114.370,-127.046,-45.960,179.786,3.953,148.690
C03416=1114.365,-126.831,-45.967,179.786,3.957,148.691
C03417=1114.360,-126.581,-45.976,179.785,3.963,148.693
C03418=1114.354,-126.331,-45.985,179.785,3.968,148.694
C03419=1114.348,-126.081,-45.993,179.785,3.973,148.695
C03420=1114.344,-125.832,-46.001,179.784,3.979,148.697
C03421=1114.339,-125.582,-46.010,179.784,3.984,148.698
C03422=1114.334,-125.332,-46.019,179.783,3.989,148.699
C03423=1114.328,-125.082,-46.027,179.783,3.996,148.701
C03424=1114.322,-124.832,-46.035,179.783,4.001,148.702
C03425=1114.317,-124.583,-46.044,179.783,4.006,148.703
C03426=1114.311,-124.333,-46.053,179.782,4.011,148.704
C03427=1114.306,-124.083,-46.061,179.781,4.017,148.706
C03428=1114.301,-123.833,-46.070,179.781,4.022,148.707
C03429=1114.296,-123.583,-46.079,179.781,4.027,148.708
C03430=1114.290,-123.334,-46.087,179.781,4.033,148.710
C03431=1114.285,-123.084,-46.096,179.780,4.038,148.711
C03432=1114.279,-122.834,-46.105,179.780,4.044,148.712
C03433=1114.274,-122.584,-46.113,179.780,4.049,148.713
C03434=1114.268,-122.335,-46.122,179.779,4.054,148.715
C03435=1114.263,-122.085,-46.131,179.779,4.060,148.716
C03436=1114.258,-121.835,-46.140,179.778,4.065,148.717
C03437=1114.253,-121.585,-46.149,179.778,4.070,148.718
C03438=1114.248,-121.335,-46.158,179.777,4.075,148.720
C03439=1114.242,-121.086,-46.165,179.777,4.081,148.721
C03440=1114.236,-120.836,-46.174,179.777,4.087,148.722
C03441=1114.231,-120.586,-46.183,179.777,4.092,148.723
C03442=1114.226,-120.336,-46.192,179.776,4.097,148.725
C03443=1114.221,-120.086,-46.201,179.776,4.102,148.726
C03444=1114.215,-119.837,-46.209,179.776,4.108,148.727
C03445=1114.210,-119.587,-46.218,179.775,4.113,148.729
C03446=1114.205,-119.337,-46.227,179.775,4.118,148.730
C03447=1114.199,-119.087,-46.237,179.774,4.123,148.731
C03448=1114.194,-118.837,-46.246,179.774,4.129,148.732
C03449=1114.188,-118.588,-46.254,179.774,4.134,148.734
C03450=1114.183,-118.338,-46.263,179.773,4.139,148.735
C03451=1114.178,-118.088,-46.272,179.773,4.144,148.736
C03452=1114.172,-117.839,-46.281,179.773,4.149,148.737
C03453=1114.167,-117.589,-46.290,179.772,4.155,148.739
C03454=1114.162,-117.339,-46.299,179.772,4.160,148.740
C03455=1114.156,-117.090,-46.307,179.772,4.165,148.741
C03456=1114.150,-116.840,-46.317,179.771,4.170,148.742
C03457=1114.145,-116.590,-46.326,179.771,4.176,148.744
C03458=1114.140,-116.340,-46.335,179.771,4.181,148.745
C03459=1114.135,-116.090,-46.343,179.770,4.186,148.746
C03460=1114.130,-115.840,-46.352,179.770,4.191,148.747
C03461=1114.125,-115.590,-46.361,179.769,4.197,148.749
C03462=1114.119,-115.340,-46.371,179.769,4.202,148.750
C03463=1114.113,-115.091,-46.379,179.769,4.207,148.751
C03464=1114.108,-114.841,-46.388,179.769,4.212,148.752
C03465=1114.104,-114.625,-46.396,179.768,4.217,148.753
C03466=1114.099,-114.410,-46.404,179.768,4.221,148.754
C03467=1114.094,-114.196,-46.412,179.768,4.225,148.755
C03468=1114.089,-113.981,-46.420,179.767,4.230,148.757
C03469=1114.085,-113.766,-46.427,179.767,4.234,148.758
C03470=1114.080,-113.550,-46.435,179.767,4.239,148.759
C03471=1114.076,-113.335,-46.443,179.766,4.243,148.760
C03472=1114.071,-113.120,-46.451,179.766,4.247,148.761
C03473=1114.066,-112.870,-46.460,179.766,4.253,148.762
C03474=1114.061,-112.621,-46.469,179.765,4.258,148.763
C03475=1114.056,-112.371,-46.478,179.765,4.263,148.765
C03476=1114.050,-112.121,-46.487,179.765,4.268,148.766
C03477=1114.045,-111.871,-46.496,179.764,4.274,148.767
C03478=1114.040,-111.621,-46.506,179.764,4.279,148.768
C03479=1114.034,-111.372,-46.514,179.764,4.284,148.769
C03480=1114.028,-111.122,-46.524,179.764,4.289,148.771
C03481=1114.023,-110.872,-46.533,179.763,4.294,148.772
C03482=1114.018,-110.622,-46.542,179.763,4.299,148.773
C03483=1114.013,-110.373,-46.551,179.763,4.305,148.774
C03484=1114.007,-110.123,-46.561,179.763,4.310,148.775
C03485=1114.002,-109.873,-46.570,179.762,4.314,148.777
C03486=1113.997,-109.623,-46.579,179.761,4.319,148.778
C03487=1113.991,-109.373,-46.588,179.761,4.324,148.779
C03488=1113.986,-109.124,-46.598,179.761,4.330,148.780
C03489=1113.981,-108.874,-46.607,179.761,4.335,148.781
C03490=1113.975,-108.624,-46.616,179.760,4.340,148.783
C03491=1113.970,-108.375,-46.626,179.760,4.345,148.784
C03492=1113.965,-108.125,-46.635,179.760,4.350,148.785
C03493=1113.959,-107.875,-46.644,179.759,4.355,148.786
C03494=1113.954,-107.625,-46.653,179.758,4.360,148.788
C03495=1113.949,-107.376,-46.663,179.758,4.365,148.789
C03496=1113.943,-107.125,-46.672,179.758,4.370,148.790
C03497=1113.938,-106.876,-46.681,179.758,4.376,148.791
C03498=1113.933,-106.626,-46.691,179.757,4.381,148.792
C03499=1113.927,-106.376,-46.700,179.757,4.386,148.794
C03500=1113.922,-106.126,-46.709,179.756,4.390,148.795
C03501=1113.917,-105.877,-46.719,179.756,4.395,148.796
C03502=1113.911,-105.627,-46.728,179.756,4.401,148.797
C03503=1113.906,-105.378,-46.738,179.756,4.406,148.798
C03504=1113.900,-105.128,-46.747,179.755,4.411,148.800
C03505=1113.895,-104.878,-46.756,179.755,4.416,148.801
C03506=1113.890,-104.628,-46.766,179.754,4.420,148.802
C03507=1113.884,-104.378,-46.775,179.754,4.426,148.803
C03508=1113.880,-104.128,-46.785,179.754,4.431,148.804
C03509=1113.874,-103.878,-46.795,179.754,4.436,148.806
C03510=1113.869,-103.628,-46.804,179.753,4.441,148.807
C03511=1113.864,-103.379,-46.813,179.753,4.446,148.808
C03512=1113.858,-103.129,-46.823,179.752,4.451,148.809
C03513=1113.853,-102.880,-46.832,179.752,4.456,148.810
C03514=1113.847,-102.630,-46.842,179.752,4.461,148.812
C03515=1113.843,-102.380,-46.851,179.752,4.466,148.813
C03516=1113.837,-102.130,-46.861,179.751,4.471,148.814
C03517=1113.832,-101.881,-46.871,179.751,4.476,148.815
C03518=1113.826,-101.631,-46.880,179.750,4.481,148.816
C03519=1113.821,-101.382,-46.890,179.751,4.485,148.817
C03520=1113.816,-101.131,-46.900,179.751,4.491,148.819
C03521=1113.811,-100.916,-46.908,179.750,4.495,148.820
C03522=1113.806,-100.701,-46.915,179.749,4.499,148.821
C03523=1113.803,-100.486,-46.924,179.749,4.503,148.822
C03524=1113.798,-100.271,-46.932,179.749,4.508,148.823
C03525=1113.792,-100.056,-46.941,179.749,4.512,148.824
C03526=1113.789,-99.841,-46.949,179.748,4.516,148.825
C03527=1113.784,-99.626,-46.957,179.748,4.520,148.826
C03528=1113.779,-99.411,-46.965,179.748,4.525,148.827
C03529=1113.773,-99.161,-46.975,179.747,4.529,148.828
C03530=1113.769,-98.911,-46.985,179.747,4.535,148.829
C03531=1113.763,-98.662,-46.995,179.747,4.540,148.831
C03532=1113.758,-98.412,-47.004,179.746,4.545,148.832
C03533=1113.753,-98.162,-47.014,179.746,4.549,148.833
C03534=1113.747,-97.912,-47.024,179.745,4.554,148.834
C03535=1113.742,-97.663,-47.033,179.746,4.559,148.835
C03536=1113.736,-97.413,-47.043,179.745,4.564,148.836
C03537=1113.732,-97.163,-47.053,179.745,4.569,148.837
C03538=1113.726,-96.913,-47.063,179.744,4.574,148.839
C03539=1113.721,-96.663,-47.072,179.744,4.579,148.840
C03540=1113.715,-96.414,-47.082,179.744,4.584,148.841
C03541=1113.710,-96.164,-47.092,179.743,4.589,148.842
C03542=1113.705,-95.914,-47.101,179.743,4.594,148.843
C03543=1113.700,-95.664,-47.112,179.743,4.599,148.845
C03544=1113.695,-95.415,-47.121,179.743,4.604,148.846
C03545=1113.689,-95.165,-47.131,179.742,4.608,148.847
C03546=1113.683,-94.915,-47.141,179.742,4.613,148.848
C03547=1113.678,-94.666,-47.151,179.741,4.619,148.849
C03548=1113.673,-94.417,-47.161,179.741,4.623,148.851
C03549=1113.668,-94.166,-47.171,179.740,4.628,148.852
C03550=1113.663,-93.916,-47.180,179.740,4.633,148.853
C03551=1113.657,-93.667,-47.191,179.739,4.638,148.854
C03552=1113.652,-93.417,-47.199,179.739,4.643,148.855
C03553=1113.647,-93.167,-47.210,179.738,4.648,148.857
C03554=1113.641,-92.917,-47.220,179.738,4.653,148.858
C03555=1113.636,-92.668,-47.230,179.737,4.657,148.859
C03556=1113.631,-92.418,-47.239,179.737,4.662,148.860
C03557=1113.625,-92.168,-47.250,179.736,4.667,148.861
C03558=1113.621,-91.918,-47.259,179.736,4.672,148.863
C03559=1113.615,-91.669,-47.270,179.735,4.676,148.864
C03560=1113.609,-91.419,-47.280,179.734,4.682,148.865
C03561=1113.604,-91.169,-47.289,179.734,4.687,148.866
C03562=1113.599,-90.919,-47.299,179.733,4.691,148.868
C03563=1113.594,-90.670,-47.310,179.733,4.696,148.869
C03564=1113.588,-90.420,-47.320,179.732,4.701,148.870
C03565=1113.583,-90.171,-47.329,179.732,4.706,148.871
C03566=1113.578,-89.920,-47.339,179.732,4.711,148.872
C03567=1113.572,-89.670,-47.349,179.731,4.716,148.874
C03568=1113.567,-89.421,-47.360,179.730,4.721,148.875
C03569=1113.562,-89.172,-47.369,179.730,4.726,148.876
C03570=1113.557,-88.921,-47.380,179.729,4.730,148.877
C03571=1113.551,-88.672,-47.390,179.729,4.735,148.879
C03572=1113.546,-88.422,-47.400,179.729,4.741,148.880
C03573=1113.541,-88.172,-47.410,179.729,4.746,148.881
C03574=1113.536,-87.922,-47.420,179.728,4.750,148.882
C03575=1113.530,-87.673,-47.430,179.727,4.756,148.883
C03576=1113.524,-87.423,-47.440,179.727,4.761,148.885
C03577=1113.518,-87.066,-47.454,179.727,4.767,148.886
C03578=1113.510,-86.709,-47.469,179.725,4.775,148.888
C03579=1113.503,-86.353,-47.484,179.725,4.782,148.890
C03580=1113.495,-85.996,-47.499,179.725,4.789,148.892
C03581=1113.490,-85.746,-47.509,179.725,4.794,148.893
C03582=1113.484,-85.496,-47.519,179.724,4.800,148.894
C03583=1113.480,-85.247,-47.529,179.724,4.805,148.895
C03584=1113.474,-84.997,-47.539,179.723,4.809,148.896
C03585=1113.469,-84.747,-47.549,179.723,4.814,148.898
C03586=1113.464,-84.497,-47.560,179.723,4.819,148.899
C03587=1113.458,-84.248,-47.570,179.723,4.824,148.900
C03588=1113.452,-83.998,-47.580,179.722,4.830,148.901
C03589=1113.448,-83.748,-47.590,179.722,4.835,148.902
C03590=1113.442,-83.499,-47.601,179.722,4.840,148.904
C03591=1113.437,-83.249,-47.611,179.721,4.845,148.905
C03592=1113.432,-82.999,-47.621,179.721,4.850,148.906
C03593=1113.426,-82.749,-47.632,179.720,4.855,148.907
C03594=1113.421,-82.500,-47.642,179.720,4.860,148.908
C03595=1113.416,-82.250,-47.652,179.720,4.865,148.910
C03596=1113.410,-82.000,-47.662,179.720,4.870,148.911
C03597=1113.406,-81.750,-47.672,179.720,4.876,148.912
C03598=1113.400,-81.501,-47.683,179.720,4.881,148.913
C03599=1113.395,-81.251,-47.693,179.719,4.886,148.914
C03600=1113.390,-81.001,-47.703,179.719,4.891,148.916
C03601=1113.384,-80.751,-47.714,179.719,4.896,148.917
C03602=1113.379,-80.501,-47.724,179.718,4.900,148.918
C03603=1113.374,-80.252,-47.735,179.718,4.906,148.919
C03604=1113.368,-80.002,-47.745,179.717,4.911,148.920
C03605=1113.363,-79.752,-47.756,179.717,4.916,148.922
C03606=1113.358,-79.503,-47.766,179.717,4.921,148.923
C03607=1113.353,-79.252,-47.777,179.717,4.927,148.924
C03608=1113.347,-79.003,-47.787,179.717,4.932,148.925
C03609=1113.341,-78.753,-47.797,179.717,4.937,148.926
C03610=1113.337,-78.504,-47.808,179.717,4.942,148.928
C03611=1113.331,-78.254,-47.819,179.716,4.947,148.929
C03612=1113.326,-78.004,-47.829,179.716,4.952,148.930
C03613=1113.319,-77.682,-47.843,179.716,4.959,148.931
C03614=1113.312,-77.358,-47.856,179.716,4.966,148.933
C03615=1113.306,-77.035,-47.870,179.716,4.973,148.934
C03616=1113.299,-76.714,-47.884,179.716,4.979,148.936
C03617=1113.294,-76.463,-47.894,179.716,4.984,148.937
C03618=1113.288,-76.214,-47.905,179.716,4.989,148.938
C03619=1113.283,-75.964,-47.915,179.716,4.994,148.939
C03620=1113.278,-75.715,-47.926,179.715,4.999,148.940
C03621=1113.273,-75.464,-47.937,179.715,5.005,148.942
C03622=1113.267,-75.215,-47.947,179.716,5.011,148.943
C03623=1113.262,-74.965,-47.957,179.716,5.016,148.944
C03624=1113.257,-74.716,-47.968,179.715,5.021,148.945
C03625=1113.251,-74.466,-47.979,179.715,5.026,148.946
C03626=1113.246,-74.216,-47.990,179.715,5.031,148.947
C03627=1113.240,-73.967,-48.001,179.715,5.036,148.949
C03628=1113.235,-73.716,-48.011,179.715,5.041,148.949
C03629=1113.231,-73.501,-48.020,179.715,5.046,148.951
C03630=1113.227,-73.287,-48.030,179.715,5.050,148.952
C03631=1113.222,-73.072,-48.039,179.715,5.055,148.953
C03632=1113.218,-72.858,-48.048,179.715,5.059,148.953
C03633=1113.213,-72.642,-48.057,179.715,5.064,148.954
C03634=1113.208,-72.427,-48.066,179.715,5.068,148.955
C03635=1113.203,-72.213,-48.076,179.715,5.073,148.956
C03636=1113.200,-71.998,-48.085,179.715,5.078,148.957
C03637=1113.194,-71.749,-48.096,179.716,5.082,148.958
C03638=1113.189,-71.498,-48.107,179.716,5.087,148.960
C03639=1113.183,-71.249,-48.118,179.716,5.093,148.961
C03640=1113.178,-70.999,-48.128,179.715,5.098,148.962
C03641=1113.173,-70.749,-48.139,179.716,5.102,148.963
C03642=1113.168,-70.500,-48.150,179.716,5.108,148.964
C03643=1113.163,-70.249,-48.160,179.716,5.114,148.965
C03644=1113.157,-70.000,-48.172,179.716,5.119,148.966
C03645=1113.152,-69.750,-48.183,179.716,5.123,148.967
C03646=1113.147,-69.501,-48.193,179.716,5.129,148.968
C03647=1113.142,-69.251,-48.204,179.716,5.134,148.970
C03648=1113.137,-69.001,-48.215,179.717,5.139,148.970
C03649=1113.131,-68.751,-48.226,179.717,5.144,148.972
C03650=1113.126,-68.502,-48.237,179.717,5.150,148.973
C03651=1113.121,-68.253,-48.248,179.717,5.154,148.974
C03652=1113.116,-68.003,-48.259,179.717,5.159,148.975
C03653=1113.110,-67.753,-48.271,179.718,5.165,148.976
C03654=1113.105,-67.503,-48.281,179.718,5.170,148.977
C03655=1113.100,-67.253,-48.292,179.718,5.175,148.978
C03656=1113.095,-67.003,-48.303,179.718,5.180,148.979
C03657=1113.089,-66.754,-48.314,179.719,5.186,148.980
C03658=1113.084,-66.504,-48.326,179.719,5.191,148.981
C03659=1113.079,-66.254,-48.336,179.719,5.196,148.982
C03660=1113.074,-66.005,-48.347,179.719,5.201,148.983
C03661=1113.068,-65.755,-48.358,179.719,5.206,148.984
C03662=1113.063,-65.506,-48.369,179.720,5.211,148.985
C03663=1113.058,-65.256,-48.381,179.720,5.217,148.986
C03664=1113.052,-65.005,-48.392,179.720,5.221,148.987
C03665=1113.048,-64.756,-48.403,179.720,5.226,148.989
C03666=1113.042,-64.507,-48.414,179.721,5.232,148.989
C03667=1113.037,-64.257,-48.426,179.722,5.237,148.990
C03668=1113.032,-64.007,-48.436,179.721,5.242,148.992
